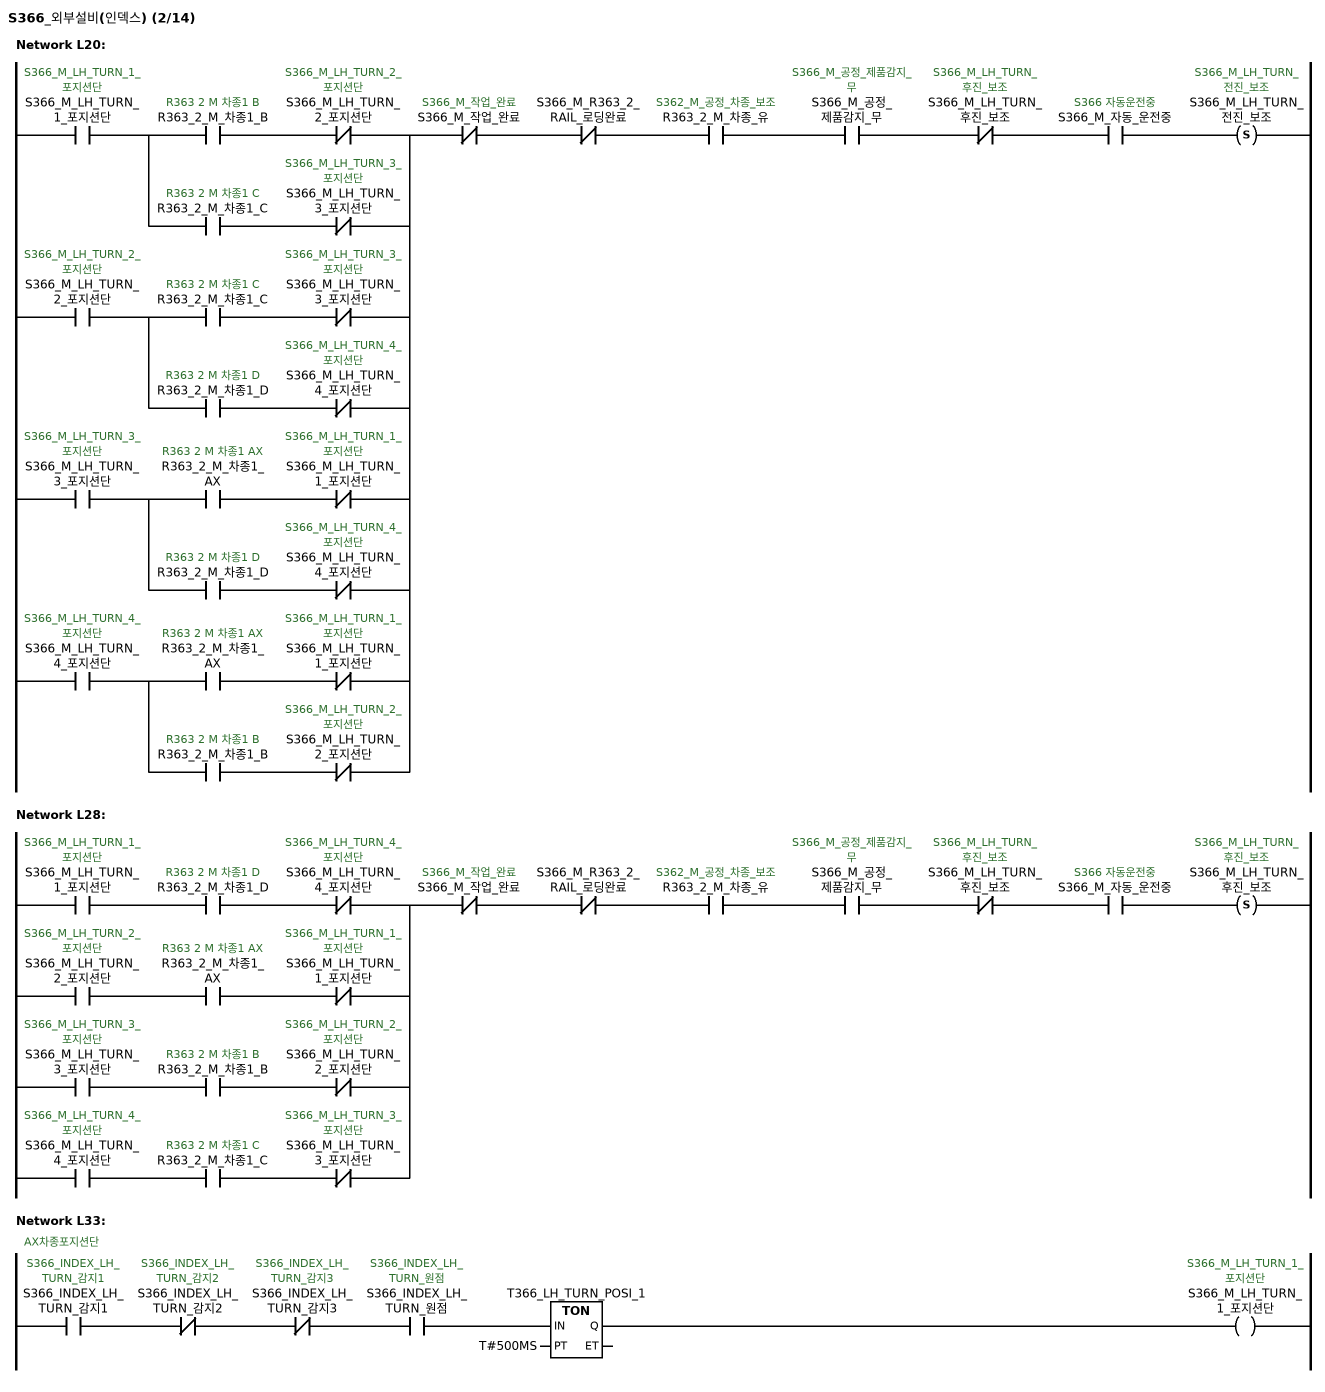
(* [picture p192: S366_외부설비(인덱스) rungs L20-L33] *)
(* Rung L20 *)
IF ((S366_M_LH_TURN_1_포지션단 AND ((R363_2_M_차종1_B AND NOT S366_M_LH_TURN_2_포지션단) OR (R363_2_M_차종1_C AND NOT S366_M_LH_TURN_3_포지션단))) OR (S366_M_LH_TURN_2_포지션단 AND ((R363_2_M_차종1_C AND NOT S366_M_LH_TURN_3_포지션단) OR (R363_2_M_차종1_D AND NOT S366_M_LH_TURN_4_포지션단))) OR (S366_M_LH_TURN_3_포지션단 AND ((R363_2_M_차종1_AX AND NOT S366_M_LH_TURN_1_포지션단) OR (R363_2_M_차종1_D AND NOT S366_M_LH_TURN_4_포지션단))) OR (S366_M_LH_TURN_4_포지션단 AND ((R363_2_M_차종1_AX AND NOT S366_M_LH_TURN_1_포지션단) OR (R363_2_M_차종1_B AND NOT S366_M_LH_TURN_2_포지션단)))) AND NOT S366_M_작업_완료 AND NOT S366_M_R363_2_RAIL_로딩완료 AND R363_2_M_차종_유 AND S366_M_공정_제품감지_무 AND NOT S366_M_LH_TURN_후진_보조 AND S366_M_자동_운전중 THEN
    S366_M_LH_TURN_전진_보조 := TRUE;
END_IF;
(* Rung L28 *)
IF ((S366_M_LH_TURN_1_포지션단 AND R363_2_M_차종1_D AND NOT S366_M_LH_TURN_4_포지션단) OR (S366_M_LH_TURN_2_포지션단 AND R363_2_M_차종1_AX AND NOT S366_M_LH_TURN_1_포지션단) OR (S366_M_LH_TURN_3_포지션단 AND R363_2_M_차종1_B AND NOT S366_M_LH_TURN_2_포지션단) OR (S366_M_LH_TURN_4_포지션단 AND R363_2_M_차종1_C AND NOT S366_M_LH_TURN_3_포지션단)) AND NOT S366_M_작업_완료 AND NOT S366_M_R363_2_RAIL_로딩완료 AND R363_2_M_차종_유 AND S366_M_공정_제품감지_무 AND NOT S366_M_LH_TURN_후진_보조 AND S366_M_자동_운전중 THEN
    S366_M_LH_TURN_후진_보조 := TRUE;
END_IF;
(* AX차종포지션단 *)
(* Rung L33 *)
T366_LH_TURN_POSI_1(IN := S366_INDEX_LH_TURN_감지1 AND NOT S366_INDEX_LH_TURN_감지2 AND NOT S366_INDEX_LH_TURN_감지3 AND S366_INDEX_LH_TURN_원점, PT := T#500MS);
S366_M_LH_TURN_1_포지션단 := T366_LH_TURN_POSI_1.Q;

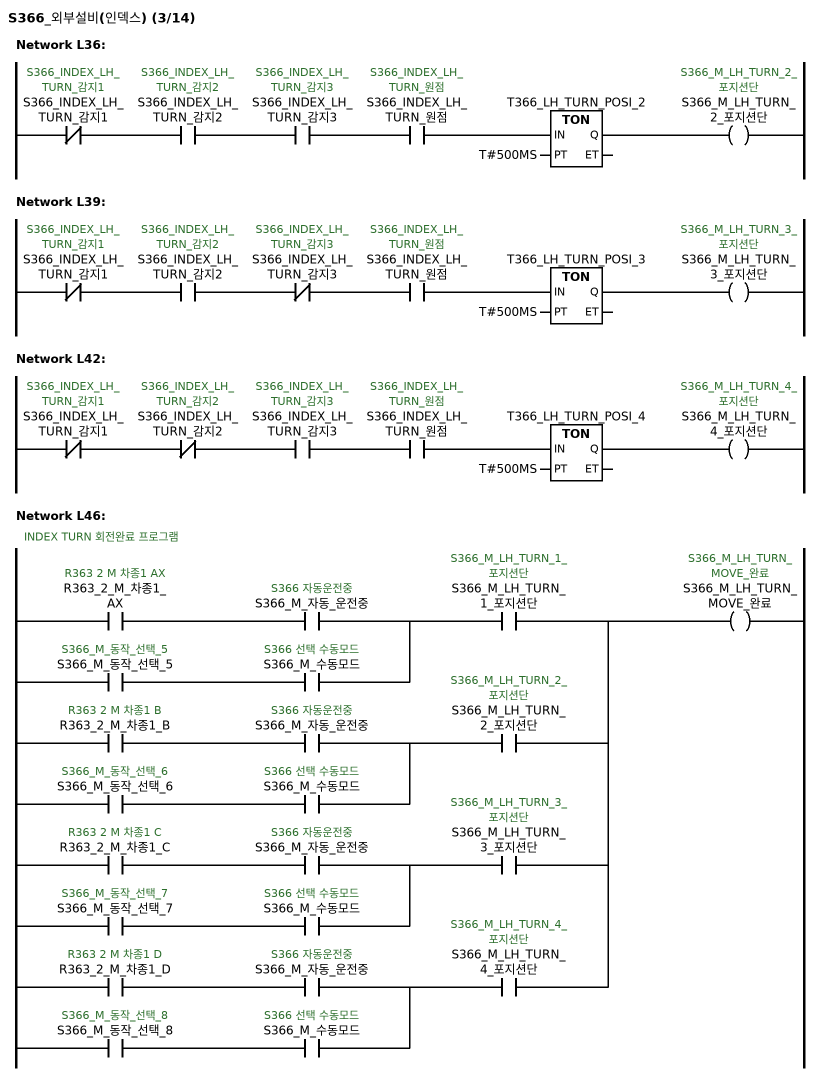
(* Rung L36 *)
T366_LH_TURN_POSI_2(IN := NOT S366_INDEX_LH_TURN_감지1 AND S366_INDEX_LH_TURN_감지2 AND S366_INDEX_LH_TURN_감지3 AND S366_INDEX_LH_TURN_원점, PT := T#500MS);
S366_M_LH_TURN_2_포지션단 := T366_LH_TURN_POSI_2.Q;
(* Rung L39 *)
T366_LH_TURN_POSI_3(IN := NOT S366_INDEX_LH_TURN_감지1 AND S366_INDEX_LH_TURN_감지2 AND NOT S366_INDEX_LH_TURN_감지3 AND S366_INDEX_LH_TURN_원점, PT := T#500MS);
S366_M_LH_TURN_3_포지션단 := T366_LH_TURN_POSI_3.Q;
(* Rung L42 *)
T366_LH_TURN_POSI_4(IN := NOT S366_INDEX_LH_TURN_감지1 AND NOT S366_INDEX_LH_TURN_감지2 AND S366_INDEX_LH_TURN_감지3 AND S366_INDEX_LH_TURN_원점, PT := T#500MS);
S366_M_LH_TURN_4_포지션단 := T366_LH_TURN_POSI_4.Q;
(* INDEX TURN 회전완료 프로그램 *)
(* Rung L46 *)
S366_M_LH_TURN_MOVE_완료 := (((R363_2_M_차종1_AX AND S366_M_자동_운전중) OR (S366_M_동작_선택_5 AND S366_M_수동모드)) AND S366_M_LH_TURN_1_포지션단) OR (((R363_2_M_차종1_B AND S366_M_자동_운전중) OR (S366_M_동작_선택_6 AND S366_M_수동모드)) AND S366_M_LH_TURN_2_포지션단) OR (((R363_2_M_차종1_C AND S366_M_자동_운전중) OR (S366_M_동작_선택_7 AND S366_M_수동모드)) AND S366_M_LH_TURN_3_포지션단) OR (((R363_2_M_차종1_D AND S366_M_자동_운전중) OR (S366_M_동작_선택_8 AND S366_M_수동모드)) AND S366_M_LH_TURN_4_포지션단);

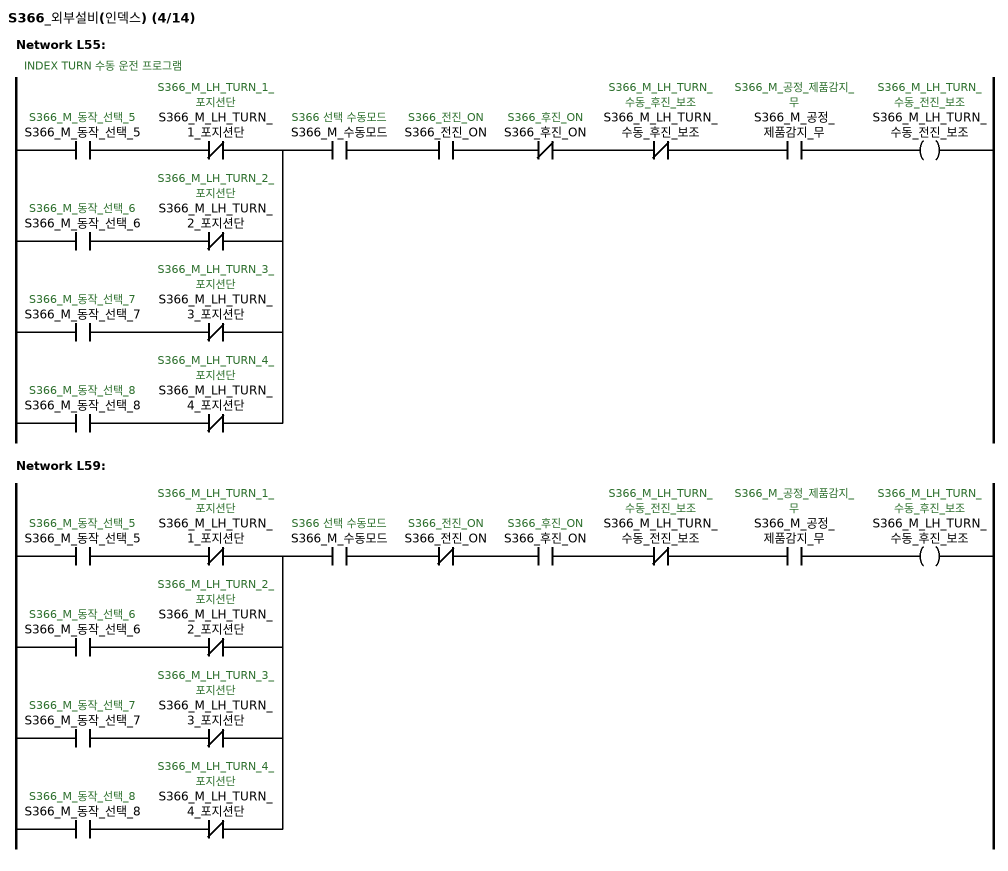
(* INDEX TURN 수동 운전 프로그램 *)
(* Rung L55 *)
S366_M_LH_TURN_수동_전진_보조 := ((S366_M_동작_선택_5 AND NOT S366_M_LH_TURN_1_포지션단) OR (S366_M_동작_선택_6 AND NOT S366_M_LH_TURN_2_포지션단) OR (S366_M_동작_선택_7 AND NOT S366_M_LH_TURN_3_포지션단) OR (S366_M_동작_선택_8 AND NOT S366_M_LH_TURN_4_포지션단)) AND S366_M_수동모드 AND S366_전진_ON AND NOT S366_후진_ON AND NOT S366_M_LH_TURN_수동_후진_보조 AND S366_M_공정_제품감지_무;
(* Rung L59 *)
S366_M_LH_TURN_수동_후진_보조 := ((S366_M_동작_선택_5 AND NOT S366_M_LH_TURN_1_포지션단) OR (S366_M_동작_선택_6 AND NOT S366_M_LH_TURN_2_포지션단) OR (S366_M_동작_선택_7 AND NOT S366_M_LH_TURN_3_포지션단) OR (S366_M_동작_선택_8 AND NOT S366_M_LH_TURN_4_포지션단)) AND S366_M_수동모드 AND NOT S366_전진_ON AND S366_후진_ON AND NOT S366_M_LH_TURN_수동_전진_보조 AND S366_M_공정_제품감지_무;

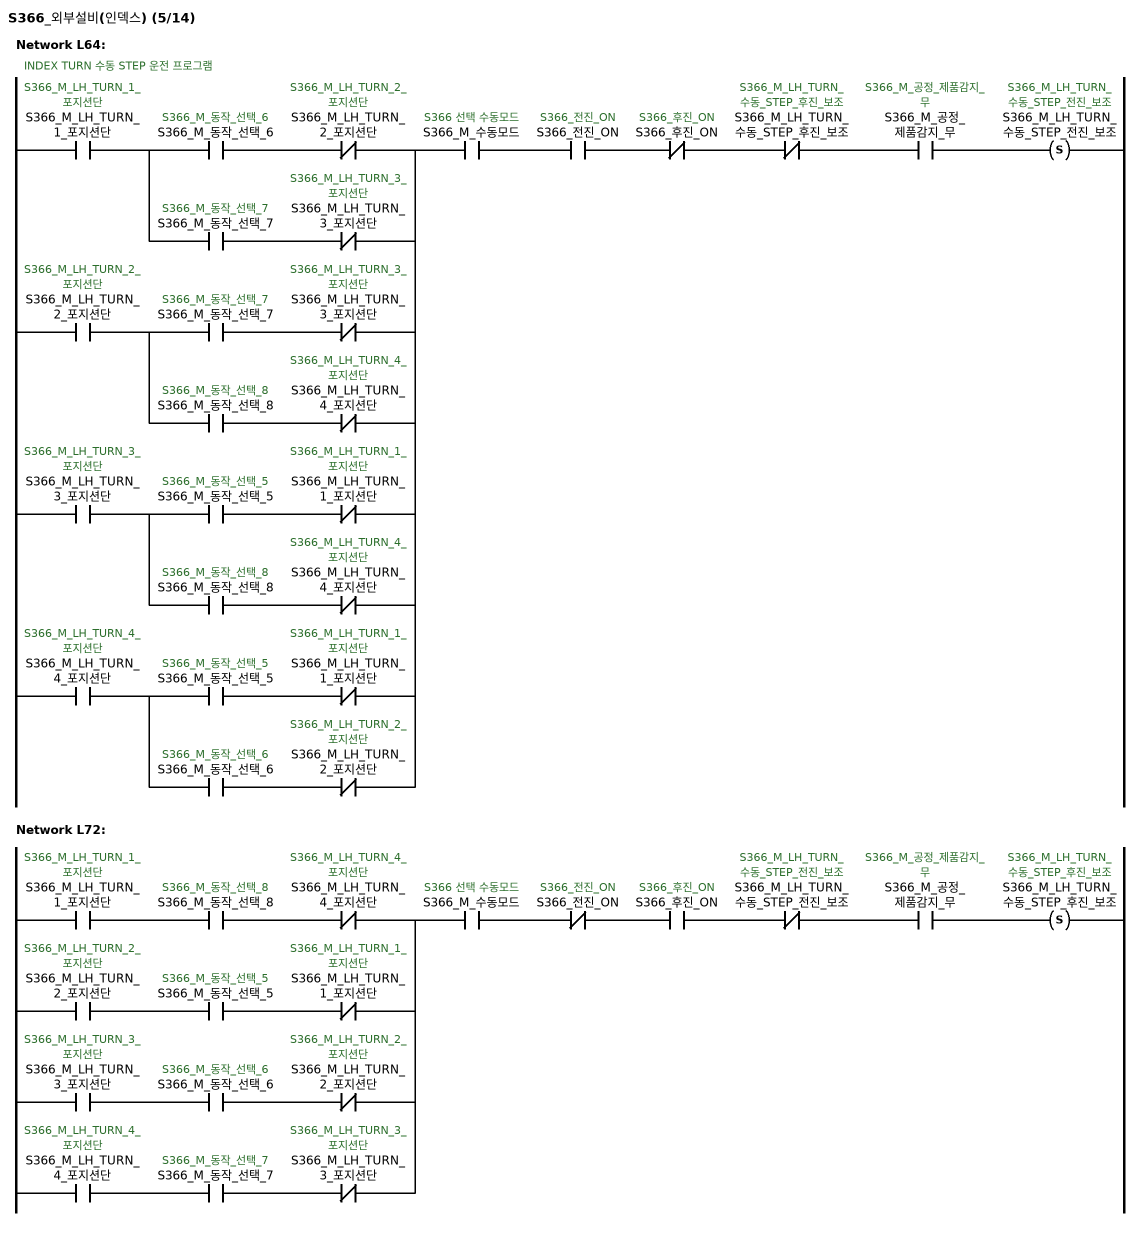
(* INDEX TURN 수동 STEP 운전 프로그램 *)
(* Rung L64 *)
IF ((S366_M_LH_TURN_1_포지션단 AND ((S366_M_동작_선택_6 AND NOT S366_M_LH_TURN_2_포지션단) OR (S366_M_동작_선택_7 AND NOT S366_M_LH_TURN_3_포지션단))) OR (S366_M_LH_TURN_2_포지션단 AND ((S366_M_동작_선택_7 AND NOT S366_M_LH_TURN_3_포지션단) OR (S366_M_동작_선택_8 AND NOT S366_M_LH_TURN_4_포지션단))) OR (S366_M_LH_TURN_3_포지션단 AND ((S366_M_동작_선택_5 AND NOT S366_M_LH_TURN_1_포지션단) OR (S366_M_동작_선택_8 AND NOT S366_M_LH_TURN_4_포지션단))) OR (S366_M_LH_TURN_4_포지션단 AND ((S366_M_동작_선택_5 AND NOT S366_M_LH_TURN_1_포지션단) OR (S366_M_동작_선택_6 AND NOT S366_M_LH_TURN_2_포지션단)))) AND S366_M_수동모드 AND S366_전진_ON AND NOT S366_후진_ON AND NOT S366_M_LH_TURN_수동_STEP_후진_보조 AND S366_M_공정_제품감지_무 THEN
    S366_M_LH_TURN_수동_STEP_전진_보조 := TRUE;
END_IF;
(* Rung L72 *)
IF ((S366_M_LH_TURN_1_포지션단 AND S366_M_동작_선택_8 AND NOT S366_M_LH_TURN_4_포지션단) OR (S366_M_LH_TURN_2_포지션단 AND S366_M_동작_선택_5 AND NOT S366_M_LH_TURN_1_포지션단) OR (S366_M_LH_TURN_3_포지션단 AND S366_M_동작_선택_6 AND NOT S366_M_LH_TURN_2_포지션단) OR (S366_M_LH_TURN_4_포지션단 AND S366_M_동작_선택_7 AND NOT S366_M_LH_TURN_3_포지션단)) AND S366_M_수동모드 AND NOT S366_전진_ON AND S366_후진_ON AND NOT S366_M_LH_TURN_수동_STEP_전진_보조 AND S366_M_공정_제품감지_무 THEN
    S366_M_LH_TURN_수동_STEP_후진_보조 := TRUE;
END_IF;

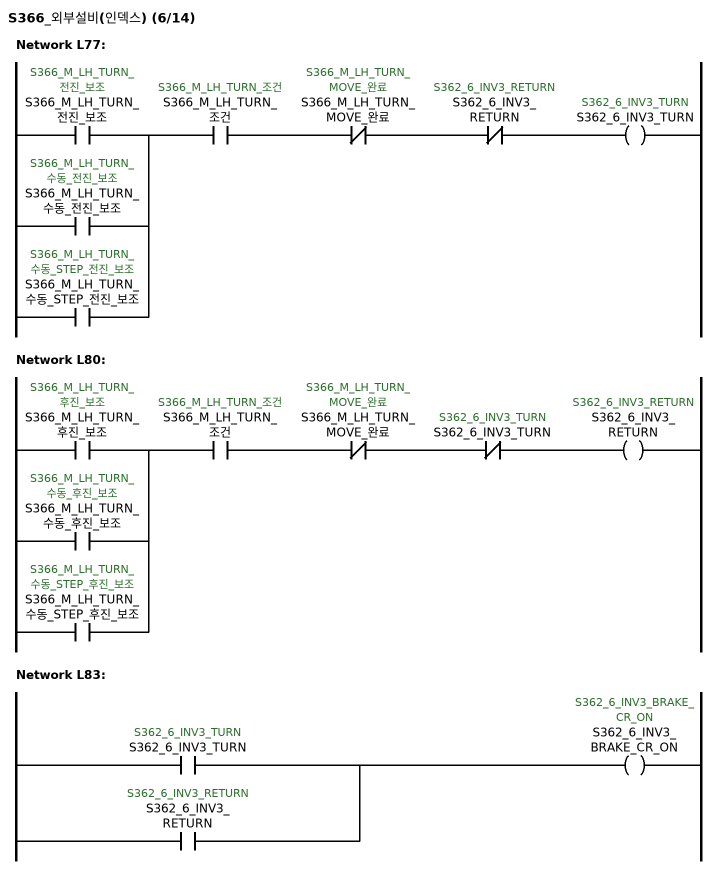
(* Rung L77 *)
S362_6_INV3_TURN := (S366_M_LH_TURN_전진_보조 OR S366_M_LH_TURN_수동_전진_보조 OR S366_M_LH_TURN_수동_STEP_전진_보조) AND S366_M_LH_TURN_조건 AND NOT S366_M_LH_TURN_MOVE_완료 AND NOT S362_6_INV3_RETURN;
(* Rung L80 *)
S362_6_INV3_RETURN := (S366_M_LH_TURN_후진_보조 OR S366_M_LH_TURN_수동_후진_보조 OR S366_M_LH_TURN_수동_STEP_후진_보조) AND S366_M_LH_TURN_조건 AND NOT S366_M_LH_TURN_MOVE_완료 AND NOT S362_6_INV3_TURN;
(* Rung L83 *)
S362_6_INV3_BRAKE_CR_ON := S362_6_INV3_TURN OR S362_6_INV3_RETURN;

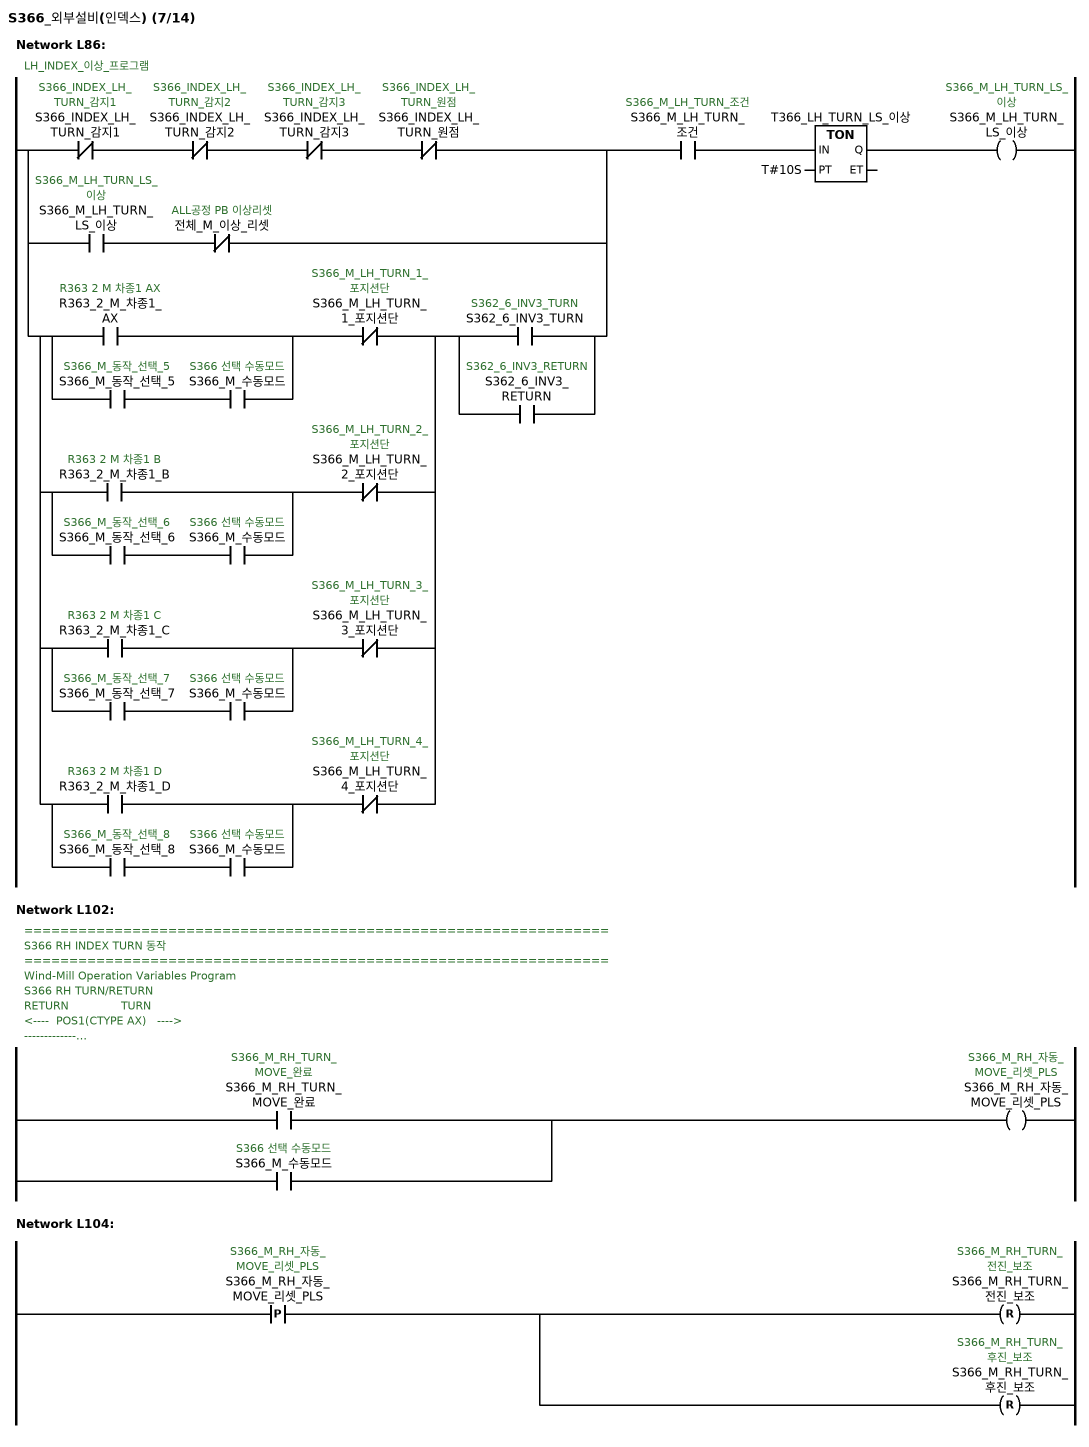
(* LH_INDEX_이상_프로그램 *)
(* Rung L86 *)
T366_LH_TURN_LS_이상(IN := ((NOT S366_INDEX_LH_TURN_감지1 AND NOT S366_INDEX_LH_TURN_감지2 AND NOT S366_INDEX_LH_TURN_감지3 AND NOT S366_INDEX_LH_TURN_원점) OR (S366_M_LH_TURN_LS_이상 AND NOT 전체_M_이상_리셋) OR ((((R363_2_M_차종1_AX OR (S366_M_동작_선택_5 AND S366_M_수동모드)) AND NOT S366_M_LH_TURN_1_포지션단) OR ((R363_2_M_차종1_B OR (S366_M_동작_선택_6 AND S366_M_수동모드)) AND NOT S366_M_LH_TURN_2_포지션단) OR ((R363_2_M_차종1_C OR (S366_M_동작_선택_7 AND S366_M_수동모드)) AND NOT S366_M_LH_TURN_3_포지션단) OR ((R363_2_M_차종1_D OR (S366_M_동작_선택_8 AND S366_M_수동모드)) AND NOT S366_M_LH_TURN_4_포지션단)) AND (S362_6_INV3_TURN OR S362_6_INV3_RETURN))) AND S366_M_LH_TURN_조건, PT := T#10S);
S366_M_LH_TURN_LS_이상 := T366_LH_TURN_LS_이상.Q;
(* ================================================================= *)
(* S366 RH INDEX TURN 동작 *)
(* ================================================================= *)
(* Wind-Mill Operation Variables Program / S366 RH TURN/RETURN *)
(* RETURN               TURN / <----  POS1(CTYPE AX)   ----> / -------------- / l              l / l              l / l              l / POS2 (CTYPE B) l              l  POS4 (CTYPE D) / l              l / l              l / l              l / -------------- / POS3 (CTYPE C) *)
(* 자동 MOVE 리셋 프로그램 *)
(* Rung L102 *)
S366_M_RH_자동_MOVE_리셋_PLS := S366_M_RH_TURN_MOVE_완료 OR S366_M_수동모드;
(* Rung L104 *)
_e3(CLK := S366_M_RH_자동_MOVE_리셋_PLS);
IF _e3.Q THEN
    S366_M_RH_TURN_전진_보조 := FALSE;
    S366_M_RH_TURN_후진_보조 := FALSE;
END_IF;

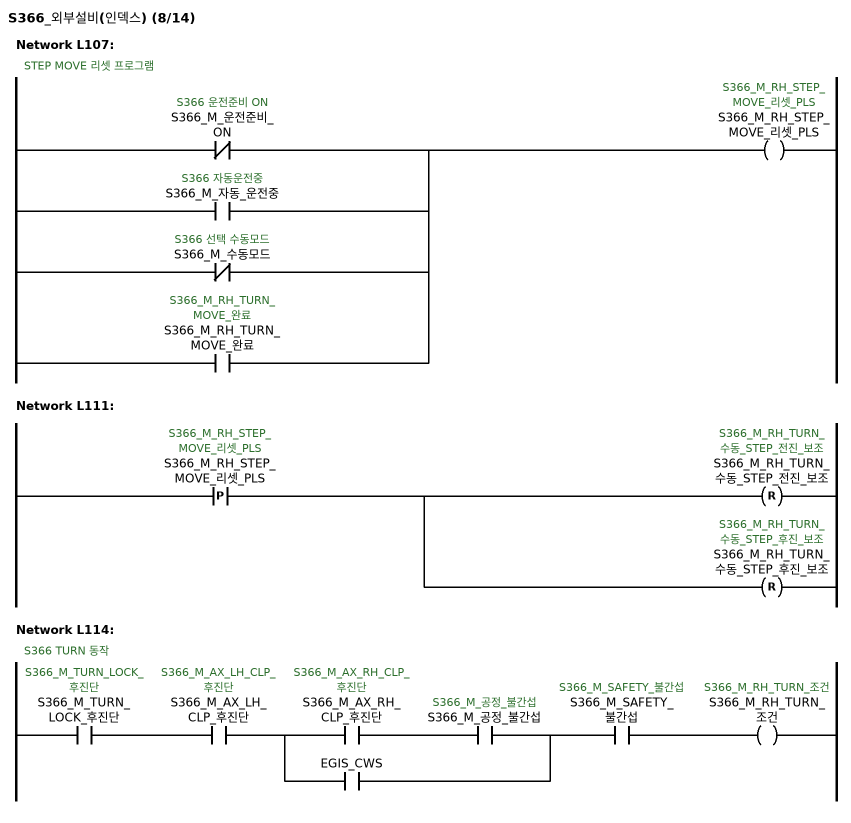
(* STEP MOVE 리셋 프로그램 *)
(* Rung L107 *)
S366_M_RH_STEP_MOVE_리셋_PLS := NOT S366_M_운전준비_ON OR S366_M_자동_운전중 OR NOT S366_M_수동모드 OR S366_M_RH_TURN_MOVE_완료;
(* Rung L111 *)
_e4(CLK := S366_M_RH_STEP_MOVE_리셋_PLS);
IF _e4.Q THEN
    S366_M_RH_TURN_수동_STEP_전진_보조 := FALSE;
    S366_M_RH_TURN_수동_STEP_후진_보조 := FALSE;
END_IF;
(* S366 TURN 동작 *)
(* Rung L114 *)
S366_M_RH_TURN_조건 := S366_M_TURN_LOCK_후진단 AND S366_M_AX_LH_CLP_후진단 AND ((S366_M_AX_RH_CLP_후진단 AND S366_M_공정_불간섭) OR EGIS_CWS) AND S366_M_SAFETY_불간섭;

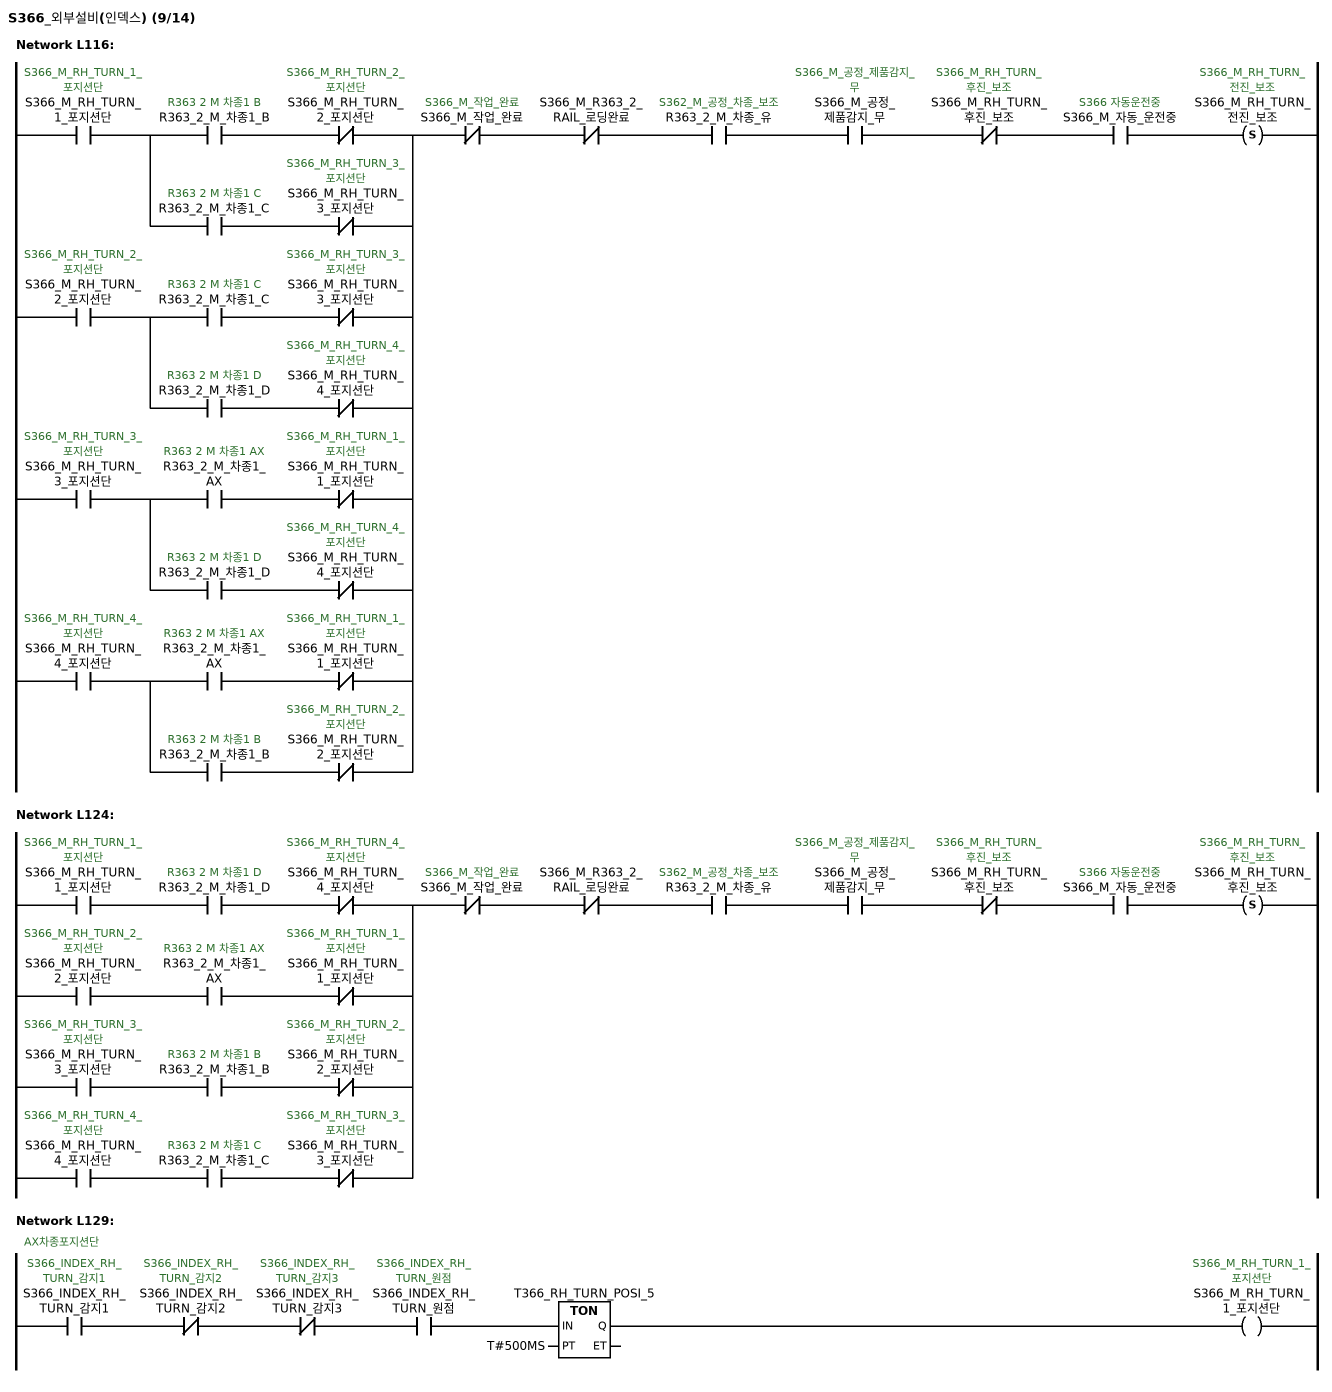
(* Rung L116 *)
IF ((S366_M_RH_TURN_1_포지션단 AND ((R363_2_M_차종1_B AND NOT S366_M_RH_TURN_2_포지션단) OR (R363_2_M_차종1_C AND NOT S366_M_RH_TURN_3_포지션단))) OR (S366_M_RH_TURN_2_포지션단 AND ((R363_2_M_차종1_C AND NOT S366_M_RH_TURN_3_포지션단) OR (R363_2_M_차종1_D AND NOT S366_M_RH_TURN_4_포지션단))) OR (S366_M_RH_TURN_3_포지션단 AND ((R363_2_M_차종1_AX AND NOT S366_M_RH_TURN_1_포지션단) OR (R363_2_M_차종1_D AND NOT S366_M_RH_TURN_4_포지션단))) OR (S366_M_RH_TURN_4_포지션단 AND ((R363_2_M_차종1_AX AND NOT S366_M_RH_TURN_1_포지션단) OR (R363_2_M_차종1_B AND NOT S366_M_RH_TURN_2_포지션단)))) AND NOT S366_M_작업_완료 AND NOT S366_M_R363_2_RAIL_로딩완료 AND R363_2_M_차종_유 AND S366_M_공정_제품감지_무 AND NOT S366_M_RH_TURN_후진_보조 AND S366_M_자동_운전중 THEN
    S366_M_RH_TURN_전진_보조 := TRUE;
END_IF;
(* Rung L124 *)
IF ((S366_M_RH_TURN_1_포지션단 AND R363_2_M_차종1_D AND NOT S366_M_RH_TURN_4_포지션단) OR (S366_M_RH_TURN_2_포지션단 AND R363_2_M_차종1_AX AND NOT S366_M_RH_TURN_1_포지션단) OR (S366_M_RH_TURN_3_포지션단 AND R363_2_M_차종1_B AND NOT S366_M_RH_TURN_2_포지션단) OR (S366_M_RH_TURN_4_포지션단 AND R363_2_M_차종1_C AND NOT S366_M_RH_TURN_3_포지션단)) AND NOT S366_M_작업_완료 AND NOT S366_M_R363_2_RAIL_로딩완료 AND R363_2_M_차종_유 AND S366_M_공정_제품감지_무 AND NOT S366_M_RH_TURN_후진_보조 AND S366_M_자동_운전중 THEN
    S366_M_RH_TURN_후진_보조 := TRUE;
END_IF;
(* AX차종포지션단 *)
(* Rung L129 *)
T366_RH_TURN_POSI_5(IN := S366_INDEX_RH_TURN_감지1 AND NOT S366_INDEX_RH_TURN_감지2 AND NOT S366_INDEX_RH_TURN_감지3 AND S366_INDEX_RH_TURN_원점, PT := T#500MS);
S366_M_RH_TURN_1_포지션단 := T366_RH_TURN_POSI_5.Q;

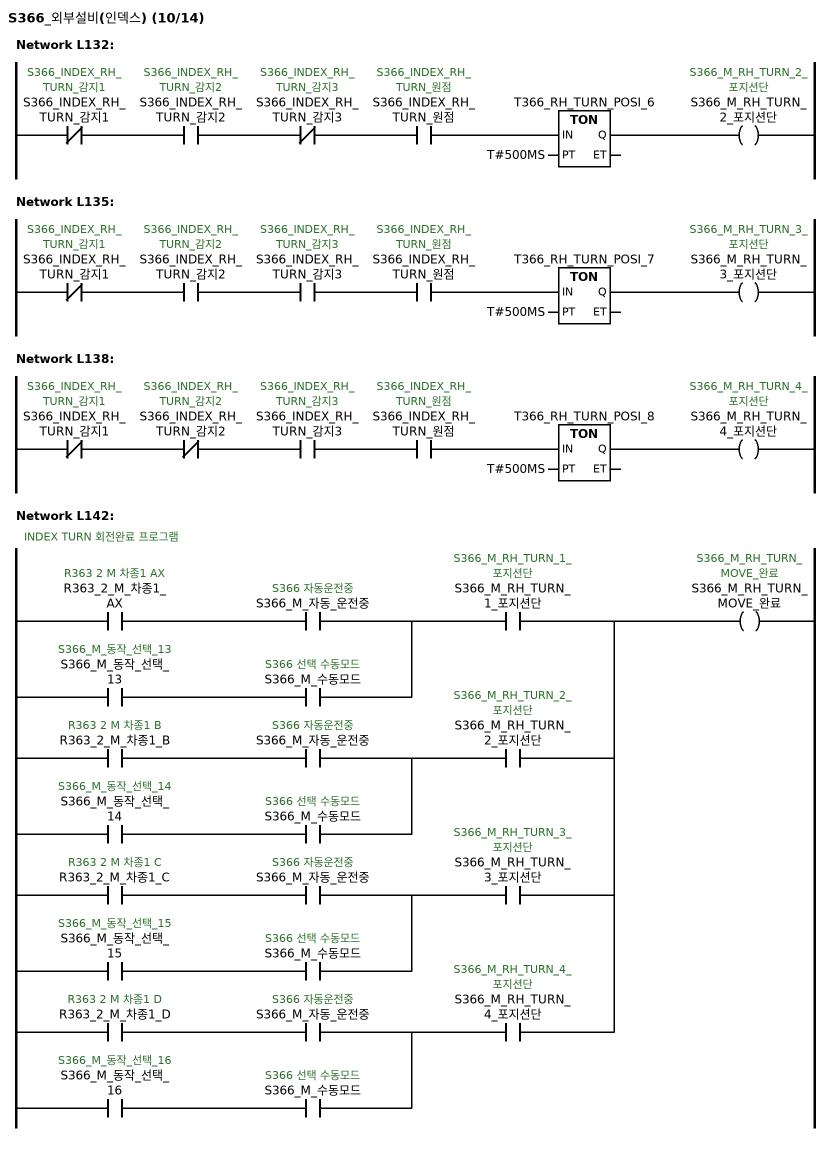
(* Rung L132 *)
T366_RH_TURN_POSI_6(IN := NOT S366_INDEX_RH_TURN_감지1 AND S366_INDEX_RH_TURN_감지2 AND NOT S366_INDEX_RH_TURN_감지3 AND S366_INDEX_RH_TURN_원점, PT := T#500MS);
S366_M_RH_TURN_2_포지션단 := T366_RH_TURN_POSI_6.Q;
(* Rung L135 *)
T366_RH_TURN_POSI_7(IN := NOT S366_INDEX_RH_TURN_감지1 AND S366_INDEX_RH_TURN_감지2 AND S366_INDEX_RH_TURN_감지3 AND S366_INDEX_RH_TURN_원점, PT := T#500MS);
S366_M_RH_TURN_3_포지션단 := T366_RH_TURN_POSI_7.Q;
(* Rung L138 *)
T366_RH_TURN_POSI_8(IN := NOT S366_INDEX_RH_TURN_감지1 AND NOT S366_INDEX_RH_TURN_감지2 AND S366_INDEX_RH_TURN_감지3 AND S366_INDEX_RH_TURN_원점, PT := T#500MS);
S366_M_RH_TURN_4_포지션단 := T366_RH_TURN_POSI_8.Q;
(* INDEX TURN 회전완료 프로그램 *)
(* Rung L142 *)
S366_M_RH_TURN_MOVE_완료 := (((R363_2_M_차종1_AX AND S366_M_자동_운전중) OR (S366_M_동작_선택_13 AND S366_M_수동모드)) AND S366_M_RH_TURN_1_포지션단) OR (((R363_2_M_차종1_B AND S366_M_자동_운전중) OR (S366_M_동작_선택_14 AND S366_M_수동모드)) AND S366_M_RH_TURN_2_포지션단) OR (((R363_2_M_차종1_C AND S366_M_자동_운전중) OR (S366_M_동작_선택_15 AND S366_M_수동모드)) AND S366_M_RH_TURN_3_포지션단) OR (((R363_2_M_차종1_D AND S366_M_자동_운전중) OR (S366_M_동작_선택_16 AND S366_M_수동모드)) AND S366_M_RH_TURN_4_포지션단);

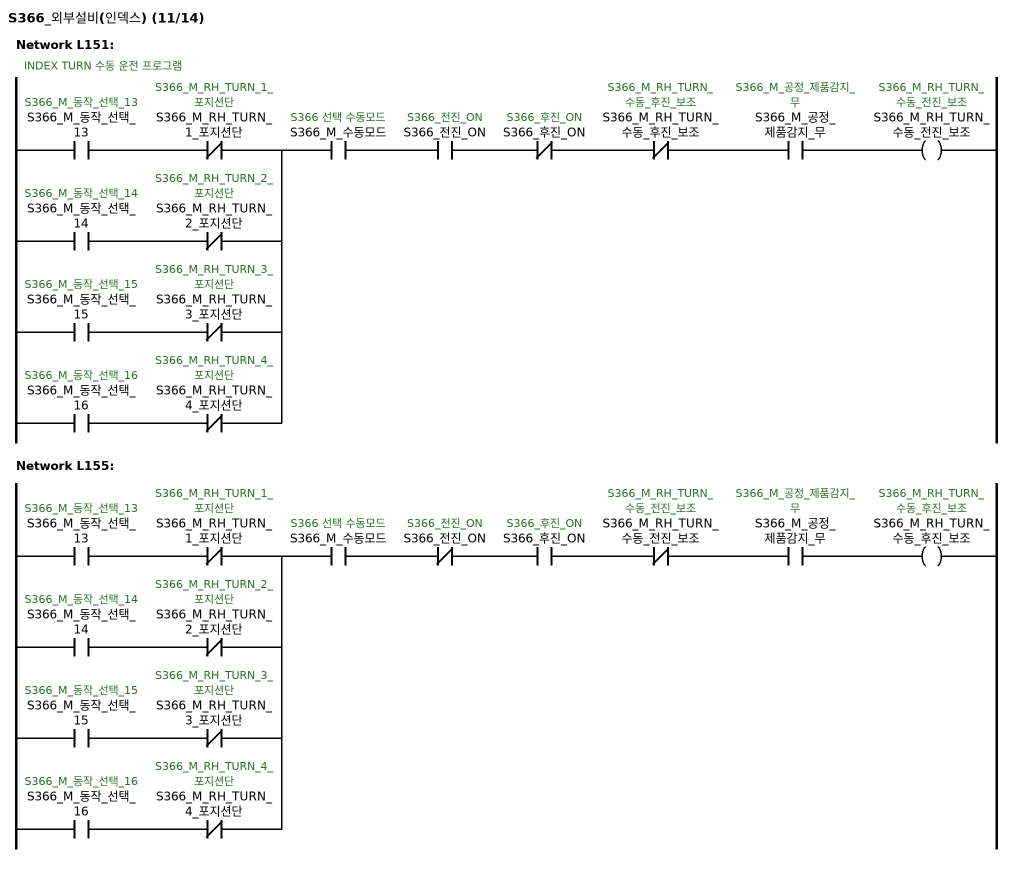
(* INDEX TURN 수동 운전 프로그램 *)
(* Rung L151 *)
S366_M_RH_TURN_수동_전진_보조 := ((S366_M_동작_선택_13 AND NOT S366_M_RH_TURN_1_포지션단) OR (S366_M_동작_선택_14 AND NOT S366_M_RH_TURN_2_포지션단) OR (S366_M_동작_선택_15 AND NOT S366_M_RH_TURN_3_포지션단) OR (S366_M_동작_선택_16 AND NOT S366_M_RH_TURN_4_포지션단)) AND S366_M_수동모드 AND S366_전진_ON AND NOT S366_후진_ON AND NOT S366_M_RH_TURN_수동_후진_보조 AND S366_M_공정_제품감지_무;
(* Rung L155 *)
S366_M_RH_TURN_수동_후진_보조 := ((S366_M_동작_선택_13 AND NOT S366_M_RH_TURN_1_포지션단) OR (S366_M_동작_선택_14 AND NOT S366_M_RH_TURN_2_포지션단) OR (S366_M_동작_선택_15 AND NOT S366_M_RH_TURN_3_포지션단) OR (S366_M_동작_선택_16 AND NOT S366_M_RH_TURN_4_포지션단)) AND S366_M_수동모드 AND NOT S366_전진_ON AND S366_후진_ON AND NOT S366_M_RH_TURN_수동_전진_보조 AND S366_M_공정_제품감지_무;

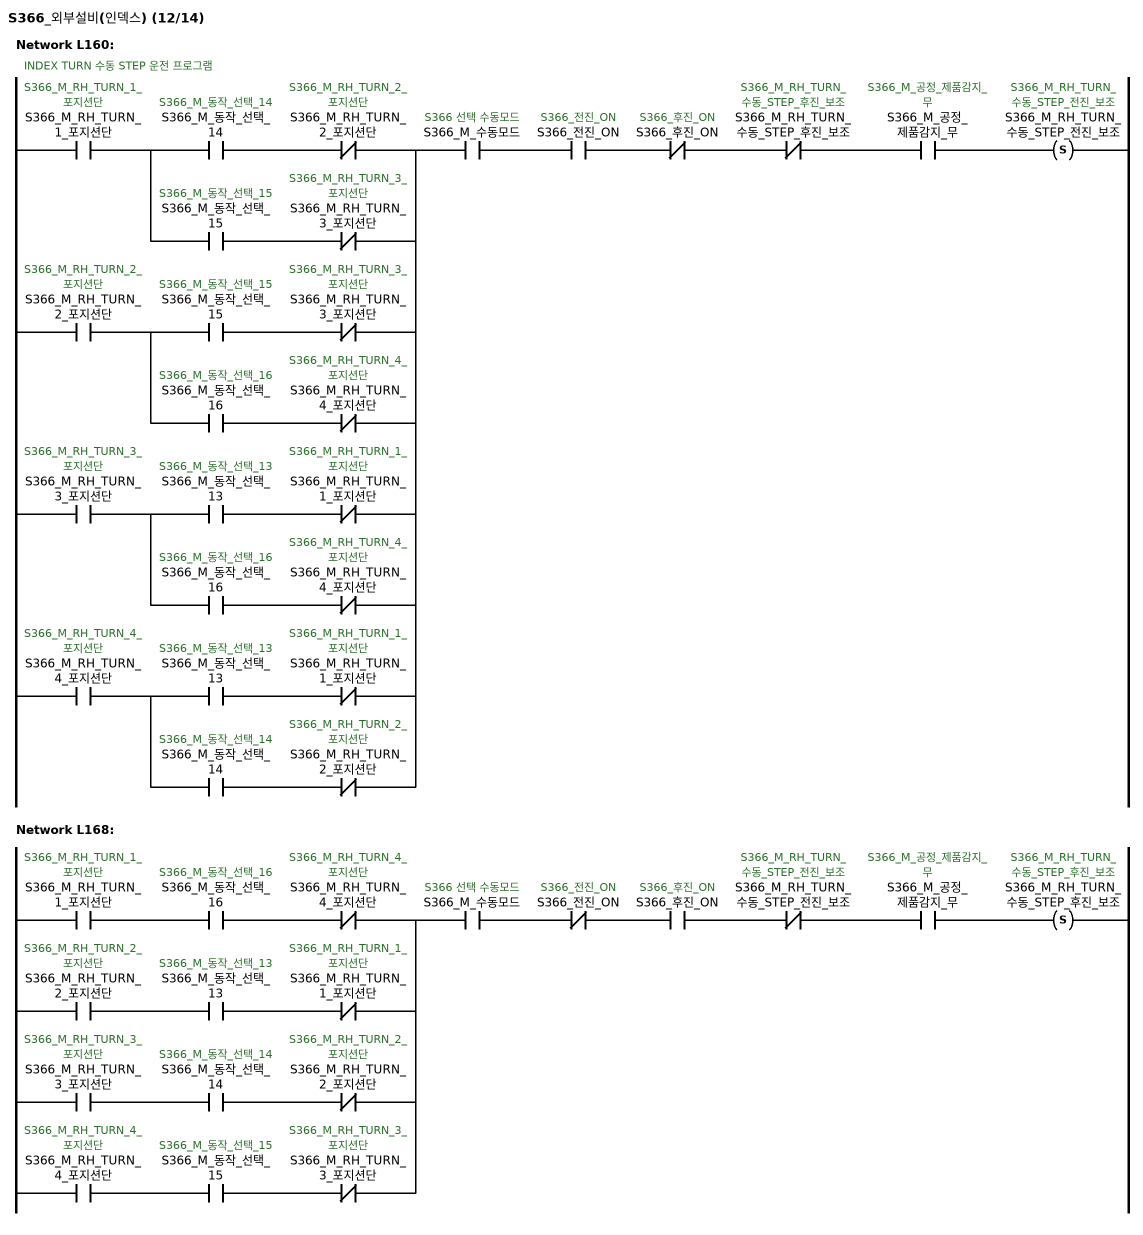
(* INDEX TURN 수동 STEP 운전 프로그램 *)
(* Rung L160 *)
IF ((S366_M_RH_TURN_1_포지션단 AND ((S366_M_동작_선택_14 AND NOT S366_M_RH_TURN_2_포지션단) OR (S366_M_동작_선택_15 AND NOT S366_M_RH_TURN_3_포지션단))) OR (S366_M_RH_TURN_2_포지션단 AND ((S366_M_동작_선택_15 AND NOT S366_M_RH_TURN_3_포지션단) OR (S366_M_동작_선택_16 AND NOT S366_M_RH_TURN_4_포지션단))) OR (S366_M_RH_TURN_3_포지션단 AND ((S366_M_동작_선택_13 AND NOT S366_M_RH_TURN_1_포지션단) OR (S366_M_동작_선택_16 AND NOT S366_M_RH_TURN_4_포지션단))) OR (S366_M_RH_TURN_4_포지션단 AND ((S366_M_동작_선택_13 AND NOT S366_M_RH_TURN_1_포지션단) OR (S366_M_동작_선택_14 AND NOT S366_M_RH_TURN_2_포지션단)))) AND S366_M_수동모드 AND S366_전진_ON AND NOT S366_후진_ON AND NOT S366_M_RH_TURN_수동_STEP_후진_보조 AND S366_M_공정_제품감지_무 THEN
    S366_M_RH_TURN_수동_STEP_전진_보조 := TRUE;
END_IF;
(* Rung L168 *)
IF ((S366_M_RH_TURN_1_포지션단 AND S366_M_동작_선택_16 AND NOT S366_M_RH_TURN_4_포지션단) OR (S366_M_RH_TURN_2_포지션단 AND S366_M_동작_선택_13 AND NOT S366_M_RH_TURN_1_포지션단) OR (S366_M_RH_TURN_3_포지션단 AND S366_M_동작_선택_14 AND NOT S366_M_RH_TURN_2_포지션단) OR (S366_M_RH_TURN_4_포지션단 AND S366_M_동작_선택_15 AND NOT S366_M_RH_TURN_3_포지션단)) AND S366_M_수동모드 AND NOT S366_전진_ON AND S366_후진_ON AND NOT S366_M_RH_TURN_수동_STEP_전진_보조 AND S366_M_공정_제품감지_무 THEN
    S366_M_RH_TURN_수동_STEP_후진_보조 := TRUE;
END_IF;

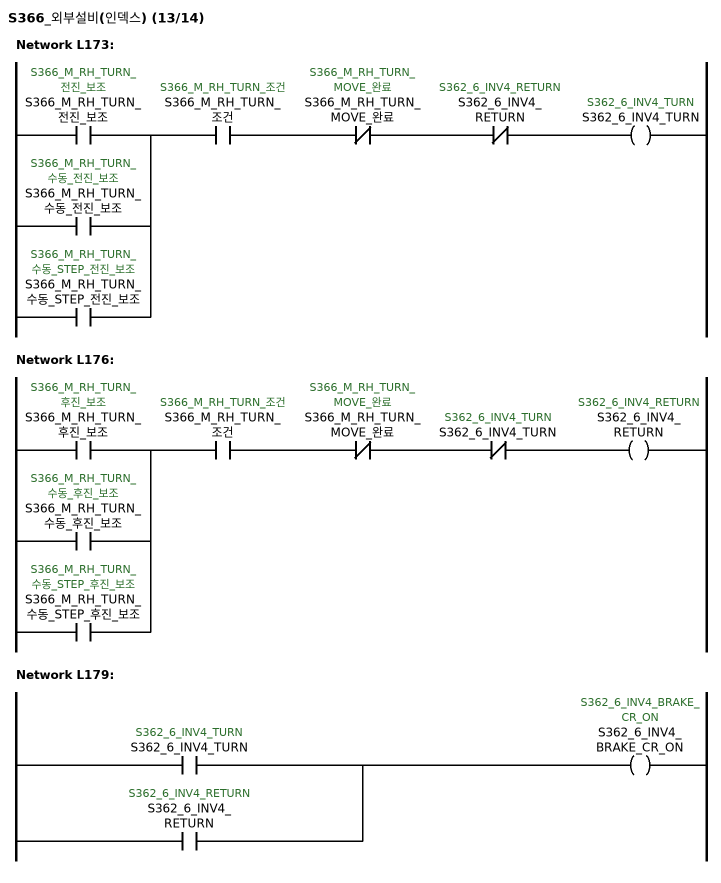
(* Rung L173 *)
S362_6_INV4_TURN := (S366_M_RH_TURN_전진_보조 OR S366_M_RH_TURN_수동_전진_보조 OR S366_M_RH_TURN_수동_STEP_전진_보조) AND S366_M_RH_TURN_조건 AND NOT S366_M_RH_TURN_MOVE_완료 AND NOT S362_6_INV4_RETURN;
(* Rung L176 *)
S362_6_INV4_RETURN := (S366_M_RH_TURN_후진_보조 OR S366_M_RH_TURN_수동_후진_보조 OR S366_M_RH_TURN_수동_STEP_후진_보조) AND S366_M_RH_TURN_조건 AND NOT S366_M_RH_TURN_MOVE_완료 AND NOT S362_6_INV4_TURN;
(* Rung L179 *)
S362_6_INV4_BRAKE_CR_ON := S362_6_INV4_TURN OR S362_6_INV4_RETURN;

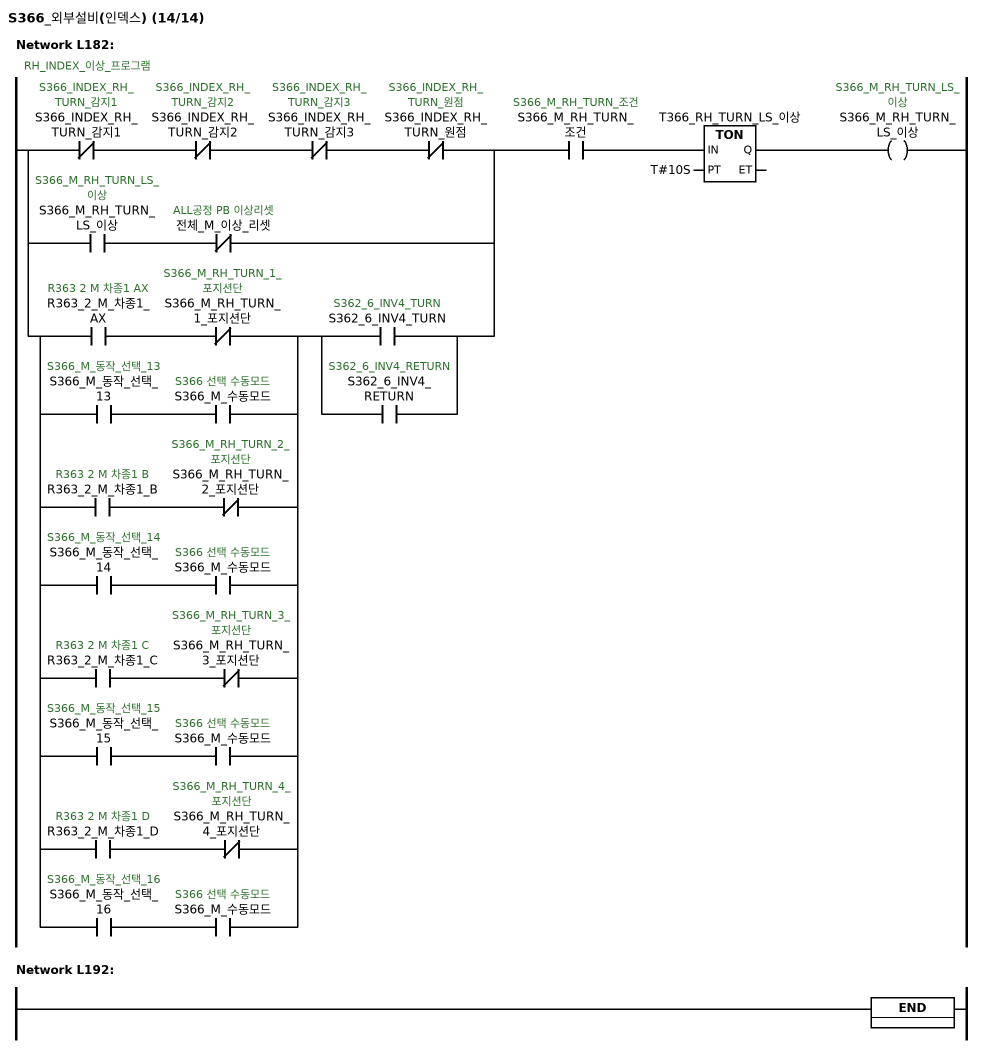
(* RH_INDEX_이상_프로그램 *)
(* Rung L182 *)
T366_RH_TURN_LS_이상(IN := ((NOT S366_INDEX_RH_TURN_감지1 AND NOT S366_INDEX_RH_TURN_감지2 AND NOT S366_INDEX_RH_TURN_감지3 AND NOT S366_INDEX_RH_TURN_원점) OR (S366_M_RH_TURN_LS_이상 AND NOT 전체_M_이상_리셋) OR (((R363_2_M_차종1_AX AND NOT S366_M_RH_TURN_1_포지션단) OR (S366_M_동작_선택_13 AND S366_M_수동모드) OR (R363_2_M_차종1_B AND NOT S366_M_RH_TURN_2_포지션단) OR (S366_M_동작_선택_14 AND S366_M_수동모드) OR (R363_2_M_차종1_C AND NOT S366_M_RH_TURN_3_포지션단) OR (S366_M_동작_선택_15 AND S366_M_수동모드) OR (R363_2_M_차종1_D AND NOT S366_M_RH_TURN_4_포지션단) OR (S366_M_동작_선택_16 AND S366_M_수동모드)) AND (S362_6_INV4_TURN OR S362_6_INV4_RETURN))) AND S366_M_RH_TURN_조건, PT := T#10S);
S366_M_RH_TURN_LS_이상 := T366_RH_TURN_LS_이상.Q;
(* Rung L192 *)
END();
END_PROGRAM

PROGRAM S366_로보트 (* task: 스캔 프로그램 *)
VAR_EXTERNAL RETAIN
    ALWAYS_ON : BOOL; (* AT %MW3.1 *) (* 항시 ON *)
    MCP_M_부저_정지 : BOOL; (* AT %MW350.5 *) (* MCP 부저정지 *)
    MCP_M_비상정지 : BOOL; (* AT %MW350.7 *) (* MCP 비상정지 이상 *)
    S366_M_R366_1_용접가능 : BOOL; (* AT %MW3004.10 *)
    S366_M_공정_제품감지_유 : BOOL; (* AT %MW3001.6 *) (* S366_M_공정_제품감지_유 *)
    S366_M_공정_차종_AX : BOOL; (* AT %MW3002.3 *) (* S366_M_공정_차종_AX *)
    S366_M_공정_차종_유 : BOOL; (* AT %MW3002.0 *) (* S366_M_공정_차종_유 *)
    S366_M_수동모드 : BOOL; (* AT %MW3000.3 *) (* S366 선택 수동모드 *)
    S366_M_자동_START : BOOL; (* AT %MW3000.5 *) (* S366 자동운전중 *)
    S366_M_자동_운전중 : BOOL; (* AT %MW3000.4 *) (* S366 자동운전중 *)
    S366_M_작업_완료 : BOOL; (* AT %MW3001.0 *) (* S366_M_작업_완료 *)
    S366_M_작업완료_SET_PLS : BOOL; (* AT %MW3000.8 *) (* S366 M 작업완료 SET PLS *)
    S366_M_작업완료_리셋_PLS : BOOL; (* AT %MW3000.9 *) (* S366 M 작업완료 리셋 PLS *)
    S366_M_차종1_AX : BOOL; (* AT %MW10161.0 *) (* S366 M 차종1 AX *)
    S366_M_총괄_이상 : BOOL; (* AT %MW3009.0 *) (* S366_M_총괄_이상 *)
    S367_M_R366_1_용접가능 : BOOL; (* AT %MW3504.9 *)
    S367_M_공정_제품감지_무 : BOOL; (* AT %MW3501.6 *) (* S367_M_공정_제품감지_무 *)
    S367_M_공정_제품감지_유 : BOOL; (* AT %MW3501.5 *) (* S367_M_공정_제품감지_유 *)
    S367_M_공정_차종_무 : BOOL; (* AT %MW3502.1 *) (* S367_M_공정_차종_무 *)
    S367_M_공정_차종_유 : BOOL; (* AT %MW3502.0 *) (* S367_M_공정_차종_유 *)
    S367_M_자동_운전중 : BOOL; (* AT %MW3500.4 *) (* S367 자동운전중 *)
    S367_M_작업_완료 : BOOL; (* AT %MW3501.0 *) (* S367_M_작업_완료 *)
    S367_M_차종1_AX : BOOL; (* AT %MW10181.0 *) (* S367 M 차종1 AX *)
    전체_M_GATE_비상정지_정상 : BOOL; (* AT %MW308.4 *) (* 전체 M GATE 비상정지 정상 *)
    전체_M_GATE_자동기동 : BOOL; (* AT %MW308.1 *) (* 전체_M_자동_운전 *)
    전체_M_운전준비_보조 : BOOL; (* AT %MW308.5 *)
    전체_M_이상_리셋 : BOOL; (* AT %MW308.2 *) (* ALL공정 PB 이상리셋 *)
    전체_공정_M_총괄_비상정지_정상 : BOOL; (* AT %MW304.1 *)
END_VAR
VAR
    INST1 : FB494_Robot_Hyundai_HMMI_v1;
    R366_1_M_RB_PROG_NO : INT;
    로보트제외 : BOOL;
END_VAR
VAR_EXTERNAL
    MCP_PBL_운전준비_ON : BOOL; (* AT %MW87630.0 *) (* MCP_PBL_운전준비_ON *)
    R361_1_M_I_RB_간섭무_1 : BOOL; (* AT %MW20012.0 *) (* R361_1_M_I_RB_간섭무_1 *)
    R363_2_M_I_RB_간섭무_1 : BOOL; (* AT %MW20042.0 *) (* R363_2_M_I_RB_간섭무_1 *)
    R366_1_I_RB_INPUT : ARRAY[0..3] OF WORD; (* AT %MW84060 *) (* R366_1_I_RB_INPUT *)
    R366_1_M_I_RB_1차_작업완료 : BOOL; (* AT %MW20061.2 *) (* R366_1_M_I_RB_1차_작업완료 *)
    R366_1_M_I_RB_2차_작업완료 : BOOL; (* AT %MW20061.3 *) (* R366_1_M_I_RB_2차_작업완료 *)
    R366_1_M_I_RB_3차_작업완료 : BOOL; (* AT %MW20061.4 *) (* R366_1_M_I_RB_3차_작업완료 *)
    R366_1_M_I_RB_4차_작업완료 : BOOL; (* AT %MW20061.5 *) (* R366_1_M_I_RB_4차_작업완료 *)
    R366_1_M_I_RB_5차_작업완료 : BOOL; (* AT %MW20061.6 *) (* R366_1_M_I_RB_5차_작업완료 *)
    R366_1_M_I_RB_6차_작업완료 : BOOL; (* AT %MW20061.7 *) (* R366_1_M_I_RB_6차_작업완료 *)
    R366_1_M_I_RB_7차_작업완료 : BOOL; (* AT %MW20061.8 *) (* R366_1_M_I_RB_7차_작업완료 *)
    R366_1_M_I_RB_PAUSE_보조 : BOOL; (* AT %MW20060.5 *) (* R366_1_M_I_RB_PAUSE_보조 *)
    R366_1_M_I_RB_PLC_RUN_CHK_이상 : BOOL; (* AT %MW20060.7 *) (* R366_1_M_I_RB_PLC_RUN_CHK_이상 *)
    R366_1_M_I_RB_간섭무_1 : BOOL; (* AT %MW20062.0 *) (* R366_1_M_I_RB_간섭무_1 *)
    R366_1_M_I_RB_간섭무_10 : BOOL; (* AT %MW20062.9 *) (* R366_1_M_I_RB_간섭무_10 *)
    R366_1_M_I_RB_간섭무_11 : BOOL; (* AT %MW20062.10 *) (* R366_1_M_I_RB_간섭무_11 *)
    R366_1_M_I_RB_간섭무_12 : BOOL; (* AT %MW20062.11 *) (* R366_1_M_I_RB_간섭무_12 *)
    R366_1_M_I_RB_간섭무_2 : BOOL; (* AT %MW20062.1 *) (* R366_1_M_I_RB_간섭무_2 *)
    R366_1_M_I_RB_간섭무_3 : BOOL; (* AT %MW20062.2 *) (* R366_1_M_I_RB_간섭무_3 *)
    R366_1_M_I_RB_간섭무_4 : BOOL; (* AT %MW20062.3 *) (* R366_1_M_I_RB_간섭무_4 *)
    R366_1_M_I_RB_간섭무_5 : BOOL; (* AT %MW20062.4 *) (* R366_1_M_I_RB_간섭무_5 *)
    R366_1_M_I_RB_간섭무_6 : BOOL; (* AT %MW20062.5 *) (* R366_1_M_I_RB_간섭무_6 *)
    R366_1_M_I_RB_간섭무_7 : BOOL; (* AT %MW20062.6 *) (* R366_1_M_I_RB_간섭무_7 *)
    R366_1_M_I_RB_간섭무_8 : BOOL; (* AT %MW20062.7 *) (* R366_1_M_I_RB_간섭무_8 *)
    R366_1_M_I_RB_간섭무_9 : BOOL; (* AT %MW20062.8 *) (* R366_1_M_I_RB_간섭무_9 *)
    R366_1_M_I_RB_비상정지 : BOOL; (* AT %MW20060.4 *) (* R366_1_M_I_RB_비상정지 *)
    R366_1_M_I_RB_운전준비 : BOOL; (* AT %MW20060.0 *) (* R366_1_M_I_RB_운전준비 *)
    R366_1_M_I_RB_원위치 : BOOL; (* AT %MW20060.3 *) (* R366_1_M_I_RB_원위치 *)
    R366_1_M_I_RB_이상 : BOOL; (* AT %MW20060.2 *) (* R366_1_M_I_RB_이상 *)
    R366_1_M_I_RB_자동 : BOOL; (* AT %MW20060.1 *) (* R366_1_M_I_RB_자동 *)
    R366_1_M_I_RB_최종작업완료 : BOOL; (* AT %MW20061.0 *) (* R366_1_M_I_RB_최종작업완료 *)
    R366_1_M_I_RB_프로그램_이상 : BOOL; (* AT %MW20060.6 *) (* R366_1_M_I_RB_프로그램_이상 *)
    R366_1_M_O_RB_1_CYCLE_SET : BOOL; (* AT %MW21060.3 *) (* R366_1_M_O_RB_1_CYCLE_SET *)
    R366_1_M_O_RB_1차_작업완료_리셋 : BOOL; (* AT %MW21062.0 *) (* R366_1_M_O_RB_1차_작업완료_리셋 *)
    R366_1_M_O_RB_2차_작업완료_리셋 : BOOL; (* AT %MW21062.1 *) (* R366_1_M_O_RB_2차_작업완료_리셋 *)
    R366_1_M_O_RB_2차_진입OK : BOOL; (* AT %MW21061.8 *) (* R366_1_M_O_RB_2차_진입OK *)
    R366_1_M_O_RB_3차_작업완료_리셋 : BOOL; (* AT %MW21062.2 *) (* R366_1_M_O_RB_3차_작업완료_리셋 *)
    R366_1_M_O_RB_3차_진입OK : BOOL; (* AT %MW21061.9 *) (* R366_1_M_O_RB_3차_진입OK *)
    R366_1_M_O_RB_4차_작업완료_리셋 : BOOL; (* AT %MW21062.3 *) (* R366_1_M_O_RB_4차_작업완료_리셋 *)
    R366_1_M_O_RB_4차_진입OK : BOOL; (* AT %MW21061.10 *) (* R366_1_M_O_RB_4차_진입OK *)
    R366_1_M_O_RB_5차_작업완료_리셋 : BOOL; (* AT %MW21062.4 *) (* R366_1_M_O_RB_5차_작업완료_리셋 *)
    R366_1_M_O_RB_5차_진입OK : BOOL; (* AT %MW21061.11 *) (* R366_1_M_O_RB_5차_진입OK *)
    R366_1_M_O_RB_6차_작업완료_리셋 : BOOL; (* AT %MW21062.5 *) (* R366_1_M_O_RB_6차_작업완료_리셋 *)
    R366_1_M_O_RB_6차_진입OK : BOOL; (* AT %MW21061.12 *) (* R366_1_M_O_RB_6차_진입OK *)
    R366_1_M_O_RB_7차_작업완료_리셋 : BOOL; (* AT %MW21062.6 *) (* R366_1_M_O_RB_7차_작업완료_리셋 *)
    R366_1_M_O_RB_7차_진입OK : BOOL; (* AT %MW21061.13 *) (* R366_1_M_O_RB_7차_진입OK *)
    R366_1_M_O_RB_ATD_OK : BOOL; (* AT %MW21060.6 *) (* R366_1_M_O_RB_ATD_OK *)
    R366_1_M_O_RB_PLT_10_진입OK : BOOL; (* AT %MW21063.10 *) (* R366_1_M_O_RB_PLT_10_진입OK *)
    R366_1_M_O_RB_PLT_11_진입OK : BOOL; (* AT %MW21063.11 *) (* R366_1_M_O_RB_PLT_11_진입OK *)
    R366_1_M_O_RB_PLT_12_진입OK : BOOL; (* AT %MW21063.12 *) (* R366_1_M_O_RB_PLT_12_진입OK *)
    R366_1_M_O_RB_PLT_1_진입OK : BOOL; (* AT %MW21063.1 *) (* R366_1_M_O_RB_PLT_1_진입OK *)
    R366_1_M_O_RB_PLT_2_진입OK : BOOL; (* AT %MW21063.2 *) (* R366_1_M_O_RB_PLT_2_진입OK *)
    R366_1_M_O_RB_PLT_3_진입OK : BOOL; (* AT %MW21063.3 *) (* R366_1_M_O_RB_PLT_3_진입OK *)
    R366_1_M_O_RB_PLT_4_진입OK : BOOL; (* AT %MW21063.4 *) (* R366_1_M_O_RB_PLT_4_진입OK *)
    R366_1_M_O_RB_PLT_5_진입OK : BOOL; (* AT %MW21063.5 *) (* R366_1_M_O_RB_PLT_5_진입OK *)
    R366_1_M_O_RB_PLT_6_진입OK : BOOL; (* AT %MW21063.6 *) (* R366_1_M_O_RB_PLT_6_진입OK *)
    R366_1_M_O_RB_PLT_7_진입OK : BOOL; (* AT %MW21063.7 *) (* R366_1_M_O_RB_PLT_7_진입OK *)
    R366_1_M_O_RB_PLT_8_진입OK : BOOL; (* AT %MW21063.8 *) (* R366_1_M_O_RB_PLT_8_진입OK *)
    R366_1_M_O_RB_PLT_9_진입OK : BOOL; (* AT %MW21063.9 *) (* R366_1_M_O_RB_PLT_9_진입OK *)
    R366_1_M_O_RB_PLT_카운터리셋_보조 : BOOL; (* AT %MW21060.10 *) (* R366_1_M_O_RB_PLT_카운터리셋_보조 *)
    R366_1_M_O_RB_PROG_NO : WORD; (* AT %MW21064 *)
    R366_1_M_O_RB_RESTART_OK : BOOL; (* AT %MW21060.2 *) (* R366_1_M_O_RB_RESTART_OK *)
    R366_1_M_O_RB_START_OK : BOOL; (* AT %MW21060.0 *) (* R366_1_M_O_RB_START_OK *)
    R366_1_M_O_RB_TEST_MODE_5000회 : BOOL; (* AT %MW21060.12 *) (* R366_1_M_O_RB_TEST_MODE_5000회 *)
    R366_1_M_O_RB_TIP_교체_시작 : BOOL; (* AT %MW21060.7 *) (* R366_1_M_O_RB_TIP_교체_시작 *)
    R366_1_M_O_RB_TIP_교체_완료 : BOOL; (* AT %MW21060.8 *) (* R366_1_M_O_RB_TIP_교체_완료 *)
    R366_1_M_O_RB_VIP_MODE : BOOL; (* AT %MW21060.11 *) (* R366_1_M_O_RB_VIP_MODE *)
    R366_1_M_O_RB_냉각수_차단_요청 : BOOL; (* AT %MW21060.9 *) (* R366_1_M_O_RB_냉각수_차단_요청 *)
    R366_1_M_O_RB_진입OK_AX차종 : BOOL; (* AT %MW21061.0 *) (* R366_1_M_O_RB_진입OK_AX차종 *)
    R366_1_M_O_RB_진입OK_B차종 : BOOL; (* AT %MW21061.1 *) (* R366_1_M_O_RB_진입OK_B차종 *)
    R366_1_M_O_RB_진입OK_C차종 : BOOL; (* AT %MW21061.2 *) (* R366_1_M_O_RB_진입OK_C차종 *)
    R366_1_M_O_RB_진입OK_D차종 : BOOL; (* AT %MW21061.3 *) (* R366_1_M_O_RB_진입OK_D차종 *)
    R366_1_M_O_RB_진입OK_E차종 : BOOL; (* AT %MW21061.4 *) (* R366_1_M_O_RB_진입OK_E차종 *)
    R366_1_M_O_RB_진입OK_F차종 : BOOL; (* AT %MW21061.5 *) (* R366_1_M_O_RB_진입OK_F차종 *)
    R366_1_M_O_RB_진입OK_G차종 : BOOL; (* AT %MW21061.6 *) (* R366_1_M_O_RB_진입OK_G차종 *)
    R366_1_M_O_RB_진입OK_H차종 : BOOL; (* AT %MW21061.7 *) (* R366_1_M_O_RB_진입OK_H차종 *)
    R366_1_M_O_RB_최종_작업완료_리셋 : BOOL; (* AT %MW21060.5 *) (* R366_1_M_O_RB_최종_작업완료_리셋 *)
    R366_1_M_O_RB_프로그램_OK : BOOL; (* AT %MW21060.1 *) (* R366_1_M_O_RB_프로그램_OK *)
    R366_1_O_RB_OUTPUT : ARRAY[0..3] OF WORD; (* AT %MW94060 *) (* R366_1_O_RB_OUTPUT *)
    R369_1_M_I_RB_간섭무_1 : BOOL; (* AT %MW20082.0 *) (* R369_1_M_I_RB_간섭무_1 *)
END_VAR
(* ladder body could not be read *)
END_PROGRAM

PROGRAM S366_로보트_용접타점수 (* task: 스캔 프로그램 *)
VAR_EXTERNAL
    R364_1_I_RB_용접타점수 : WORD; (* AT %MW84055 *) (* R364_1_I_RB_용접타점수 *)
    R364_1_M_I_RB_1차_작업완료 : BOOL; (* AT %MW20051.2 *) (* R364_1_M_I_RB_1차_작업완료 *)
    R366_1_I_RB_용접타점수 : WORD; (* AT %MW84065 *) (* R366_1_I_RB_용접타점수 *)
END_VAR
VAR_EXTERNAL RETAIN
    R364_1_M_AX_차종_용접타점수 : WORD; (* AT %MW8010 *)
    R364_1_M_용접완료 : BOOL; (* AT %MW2006.1 *)
    R364_1_M_용접타점수_OK : BOOL; (* AT %MW2006.8 *)
    R366_1_M_용접완료 : BOOL; (* AT %MW3006.1 *)
    R366_1_M_용접타점수_OK : BOOL; (* AT %MW3006.8 *)
    S364_M_전체_용접완료 : BOOL; (* AT %MW2006.0 *)
    S366_M_R366_1_용접완료 : BOOL; (* AT %MW3001.3 *)
    S366_M_전체_용접완료 : BOOL; (* AT %MW3006.0 *)
    S366_M_차종1_AX : BOOL; (* AT %MW10161.0 *) (* S366 M 차종1 AX *)
END_VAR
VAR
    _t1 : BOOL;
END_VAR

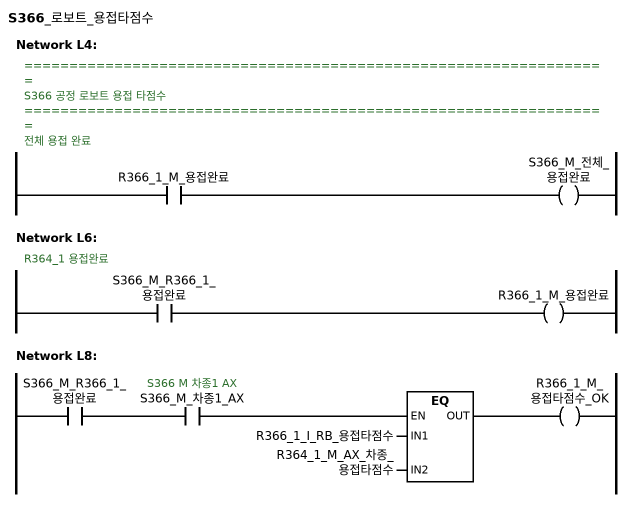
(* ================================================================= *)
(* S366 공정 로보트 용접 타점수 *)
(* ================================================================= *)
(* 전체 용접 완료 *)
(* Rung L4 *)
S366_M_전체_용접완료 := R366_1_M_용접완료;
(* R364_1 용접완료 *)
(* Rung L6 *)
R366_1_M_용접완료 := S366_M_R366_1_용접완료;
(* Rung L8 *)
IF S366_M_R366_1_용접완료 AND S366_M_차종1_AX THEN _t1 := R366_1_I_RB_용접타점수 = R364_1_M_AX_차종_용접타점수; END_IF;
R366_1_M_용접타점수_OK := _t1;
END_PROGRAM

PROGRAM S366_이상 (* task: 스캔 프로그램 *)
VAR
    INST : TON;
    INST1 : TON;
    INST10 : TON;
    INST11 : TON;
    INST12 : TON;
    INST13 : TON;
    INST14 : TON;
    INST15 : TON;
    INST16 : TON;
    INST17 : TON;
    INST18 : TON;
    INST19 : TON;
    INST2 : TON;
    INST20 : TON;
    INST21 : TON;
    INST22 : TON;
    INST23 : TON;
    INST24 : TON;
    INST25 : TON;
    INST26 : TON;
    INST27 : TON;
    INST28 : TON;
    INST29 : TON;
    INST3 : TON;
    INST30 : TON;
    INST31 : TON;
    INST32 : TON;
    INST33 : TON;
    INST34 : TON;
    INST35 : TON;
    INST36 : TON;
    INST37 : TON;
    INST38 : TON;
    INST39 : TON;
    INST4 : TON;
    INST40 : TON;
    INST41 : TON;
    INST42 : TON;
    INST43 : TON;
    INST5 : TON;
    INST6 : TON;
    INST7 : TON;
    INST8 : TON;
    INST9 : TON;
    T366_LH_TURN_LS_이상 : TON;
    T366_RH_TURN_LS_이상 : TON;
END_VAR
VAR_EXTERNAL
    R361_1_M_I_RB_이상 : BOOL; (* AT %MW20010.2 *) (* R361_1_M_I_RB_이상 *)
    R361_1_M_I_RB_프로그램_이상 : BOOL; (* AT %MW20010.6 *) (* R361_1_M_I_RB_프로그램_이상 *)
    R366_1_M_I_RB_이상 : BOOL; (* AT %MW20060.2 *) (* R366_1_M_I_RB_이상 *)
    R366_1_M_I_RB_프로그램_이상 : BOOL; (* AT %MW20060.6 *) (* R366_1_M_I_RB_프로그램_이상 *)
    S362_6_INV1_NFB_ON : BOOL; (* AT %MW85013.0 *) (* S362_6_INV1_NFB_ON *)
    S362_6_INV1_NOMAL_OK : BOOL; (* AT %MW85010.0 *) (* S362_6_INV1_NOMAL_OK *)
    S362_6_INV3_BRAKE_CR_ON : BOOL; (* AT %MW95015.7 *) (* S362_6_INV3_BRAKE_CR_ON *)
    S362_6_INV3_MC_BRAKE_ON : BOOL; (* AT %MW85010.9 *) (* S362_6_INV3_MC_BRAKE_ON *)
    S362_6_INV3_NFB_ON : BOOL; (* AT %MW85013.2 *) (* S362_6_INV3_NFB_ON *)
    S362_6_INV3_NOMAL_OK : BOOL; (* AT %MW85010.8 *) (* S362_6_INV3_NOMAL_OK *)
    S362_6_INV3_RETURN : BOOL; (* AT %MW95015.1 *) (* S362_6_INV3_RETURN *)
    S362_6_INV3_TURN : BOOL; (* AT %MW95015.0 *) (* S362_6_INV3_TURN *)
    S362_6_INV4_BRAKE_CR_ON : BOOL; (* AT %MW95015.15 *) (* S362_6_INV4_BRAKE_CR_ON *)
    S362_6_INV4_MC_BRAKE_ON : BOOL; (* AT %MW85010.13 *) (* S362_6_INV4_MC_BRAKE_ON *)
    S362_6_INV4_NFB_ON : BOOL; (* AT %MW85013.3 *) (* S362_6_INV4_NFB_ON *)
    S362_6_INV4_NOMAL_OK : BOOL; (* AT %MW85010.12 *) (* S362_6_INV4_NOMAL_OK *)
    S362_6_INV4_RETURN : BOOL; (* AT %MW95015.9 *) (* S362_6_INV4_RETURN *)
    S362_6_INV4_TURN : BOOL; (* AT %MW95015.8 *) (* S362_6_INV4_TURN *)
    S366R_8_10_PLC_BOX_CP_TRIP : BOOL; (* AT %MW88100.15 *) (* S366L_LS_AX_MAINTENANCE_CHK *)
    S366R_8_20_PLC_BOX_CP_TRIP : BOOL; (* AT %MW88200.15 *) (* S366R_LS_AX_MAINTENANCE_CHK *)
    S366_6_10_PLC_BOX_CP_TRIP : BOOL; (* AT %MW86102.15 *) (* S366_6_10_PLC_BOX_CP_TRIP *)
    S366_INDEX_LH_TURN_감지1 : BOOL; (* AT %MW86101.4 *) (* S366_INDEX_LH_TURN_감지1 *)
    S366_INDEX_LH_TURN_감지2 : BOOL; (* AT %MW86101.5 *) (* S366_INDEX_LH_TURN_감지2 *)
    S366_INDEX_LH_TURN_감지3 : BOOL; (* AT %MW86101.6 *) (* S366_INDEX_LH_TURN_감지3 *)
    S366_INDEX_LH_TURN_원점 : BOOL; (* AT %MW86101.7 *) (* S366_INDEX_LH_TURN_원점 *)
    S366_INDEX_RH_TURN_감지1 : BOOL; (* AT %MW86101.0 *) (* S366_INDEX_RH_TURN_감지1 *)
    S366_INDEX_RH_TURN_감지2 : BOOL; (* AT %MW86101.1 *) (* S366_INDEX_RH_TURN_감지2 *)
    S366_INDEX_RH_TURN_감지3 : BOOL; (* AT %MW86101.2 *) (* S366_INDEX_RH_TURN_감지3 *)
    S366_INDEX_RH_TURN_원점 : BOOL; (* AT %MW86101.3 *) (* S366_INDEX_RH_TURN_원점 *)
    S366_LH_CUT_OFF_BOX_ON : BOOL; (* AT %MW86102.10 *)
    S366_RH_CUT_OFF_BOX_ON : BOOL; (* AT %MW86102.11 *)
    S366_공기압_AIR_CHECK : BOOL; (* AT %MW86102.14 *) (* S366_공기압_AIR_CHECK *)
    _0004_EB05_CFG_ER : BOOL; (* AT %MW184032.0 *) (* EB 구성 에러 *)
    _0004_EB05_DEER : BOOL; (* AT %MW184032.1 *) (* EB 운전 중 탈락 *)
    _0004_EB06_CFG_ER : BOOL; (* AT %MW184034.8 *) (* EB 구성 에러 *)
    _0004_EB06_DEER : BOOL; (* AT %MW184034.9 *) (* EB 운전 중 탈락 *)
    _0006_EB10_CFG_ER : BOOL; (* AT %MW186028.0 *) (* EB 구성 에러 *)
    _0006_EB10_DEER : BOOL; (* AT %MW186028.1 *) (* EB 운전 중 탈락 *)
    _0006_EB10_IO_DEER : BOOL; (* AT %MW186029.2 *) (* EB IO 탈락 에러 *)
    _0006_EB10_IO_TYER : BOOL; (* AT %MW186029.1 *) (* EB IO 타입 에러 *)
    _0006_EB41_CFG_ER : BOOL; (* AT %MW186064.0 *) (* EB 구성 에러 *)
    _0006_EB41_DEER : BOOL; (* AT %MW186064.1 *) (* EB 운전 중 탈락 *)
    _0006_EB41_IO_DEER : BOOL; (* AT %MW186065.2 *) (* EB IO 탈락 에러 *)
    _0006_EB41_IO_TYER : BOOL; (* AT %MW186065.1 *) (* EB IO 타입 에러 *)
END_VAR
VAR_EXTERNAL RETAIN
    R366_1_M_NODE_4_06_통신_이상 : BOOL; (* AT %MW3024.8 *)
    R366_1_M_용접_카운트_이상 : BOOL; (* AT %MW3029.0 *)
    R366_1_M_용접타점수_OK : BOOL; (* AT %MW3006.8 *)
    S362_M_공정_불간섭 : BOOL; (* AT %MW1004.1 *) (* S362_M_공정_불간섭 *)
    S362_M_공정_제품감지_무 : BOOL; (* AT %MW1001.5 *) (* S362_M_공정_제품감지_무 *)
    S362_M_공정_차종_유 : BOOL; (* AT %MW1002.0 *) (* S362_M_공정_차종_유 *)
    S362_M_자동_운전중 : BOOL; (* AT %MW1000.4 *) (* S362 자동운전중 *)
    S366_LH_M_NODE_8_10_통신_이상 : BOOL; (* AT %MW3024.1 *)
    S366_M_AX_LH_CLP_전진_LS_이상 : BOOL; (* AT %MW3104.5 *) (* S366_M_AX_LH_CLP_전진_LS_이상 *)
    S366_M_AX_LH_CLP_후진_LS_이상 : BOOL; (* AT %MW3104.6 *) (* S366_M_AX_LH_CLP_후진_LS_이상 *)
    S366_M_AX_RH_CLP_전진_LS_이상 : BOOL; (* AT %MW3112.5 *) (* S366_M_AX_RH_CLP_전진_LS_이상 *)
    S366_M_AX_RH_CLP_후진_LS_이상 : BOOL; (* AT %MW3112.6 *) (* S366_M_AX_RH_CLP_후진_LS_이상 *)
    S366_M_CP_OFF : BOOL; (* AT %MW3017.0 *)
    S366_M_LH_CB_OFF : BOOL; (* AT %MW3021.2 *)
    S366_M_LH_CP_OFF : BOOL; (* AT %MW3017.2 *) (* S366_M_LH_CP_OFF *)
    S366_M_LH_INV_이상 : BOOL; (* AT %MW3019.0 *) (* S366_M_LH_INV_이상 *)
    S366_M_LH_MC_이상 : BOOL; (* AT %MW3023.0 *) (* S366_M_LH_MC_이상 *)
    S366_M_LH_NFB_OFF : BOOL; (* AT %MW3021.0 *) (* S366_M_LH_NFB_OFF *)
    S366_M_LH_TURN_1_포지션단 : BOOL; (* AT %MW3101.3 *) (* S366_M_LH_TURN_1_포지션단 *)
    S366_M_LH_TURN_2_포지션단 : BOOL; (* AT %MW3101.4 *) (* S366_M_LH_TURN_2_포지션단 *)
    S366_M_LH_TURN_3_포지션단 : BOOL; (* AT %MW3101.5 *) (* S366_M_LH_TURN_3_포지션단 *)
    S366_M_LH_TURN_4_포지션단 : BOOL; (* AT %MW3101.6 *) (* S366_M_LH_TURN_4_포지션단 *)
    S366_M_LH_TURN_LS_이상 : BOOL; (* AT %MW3101.7 *) (* S366_M_LH_TURN_LS_이상 *)
    S366_M_LH_TURN_조건 : BOOL; (* AT %MW3101.0 *) (* S366_M_LH_TURN_조건 *)
    S366_M_NODE_6_10_통신_이상 : BOOL; (* AT %MW3024.0 *)
    S366_M_R361_1_ROOF_로딩완료 : BOOL; (* AT %MW3001.2 *)
    S366_M_R361_1_동일차종_OK : BOOL; (* AT %MW3005.8 *)
    S366_M_R361_1_차종매칭_조건 : BOOL; (* AT %MW3005.0 *)
    S366_M_R363_2_RAIL_로딩완료 : BOOL; (* AT %MW3001.1 *)
    S366_M_R366_1_용접완료 : BOOL; (* AT %MW3001.3 *)
    S366_M_RH_CB_OFF : BOOL; (* AT %MW3021.3 *)
    S366_M_RH_CP_OFF : BOOL; (* AT %MW3017.3 *) (* S366_M_RH_CP_OFF *)
    S366_M_RH_INV_이상 : BOOL; (* AT %MW3019.1 *) (* S366_M_RH_INV_이상 *)
    S366_M_RH_MC_이상 : BOOL; (* AT %MW3023.1 *) (* S366_M_RH_MC_이상 *)
    S366_M_RH_NFB_OFF : BOOL; (* AT %MW3021.1 *) (* S366_M_RH_NFB_OFF *)
    S366_M_RH_TURN_1_포지션단 : BOOL; (* AT %MW3109.3 *) (* S366_M_RH_TURN_1_포지션단 *)
    S366_M_RH_TURN_2_포지션단 : BOOL; (* AT %MW3109.4 *) (* S366_M_RH_TURN_2_포지션단 *)
    S366_M_RH_TURN_3_포지션단 : BOOL; (* AT %MW3109.5 *) (* S366_M_RH_TURN_3_포지션단 *)
    S366_M_RH_TURN_4_포지션단 : BOOL; (* AT %MW3109.6 *) (* S366_M_RH_TURN_4_포지션단 *)
    S366_M_RH_TURN_LS_이상 : BOOL; (* AT %MW3109.7 *) (* S366_M_RH_TURN_LS_이상 *)
    S366_M_RH_TURN_조건 : BOOL; (* AT %MW3109.0 *) (* S366_M_RH_TURN_조건 *)
    S366_M_SAFETY_불간섭 : BOOL; (* AT %MW3004.4 *) (* S366_M_SAFETY_불간섭 *)
    S366_M_TURN_LOCK_전진_LS_이상 : BOOL; (* AT %MW3100.5 *) (* S366_M_TURN_LOCK_전진_LS_이상 *)
    S366_M_TURN_LOCK_후진_LS_이상 : BOOL; (* AT %MW3100.6 *) (* S366_M_TURN_LOCK_후진_LS_이상 *)
    S366_M_공정_AX_FRT_PNL_제품감지_이상 : BOOL; (* AT %MW3014.4 *)
    S366_M_공정_AX_RAIL_제품감지_이상 : BOOL; (* AT %MW3014.3 *)
    S366_M_공정_AX_RR_PNL_제품감지_이상 : BOOL; (* AT %MW3014.5 *)
    S366_M_공정_AX_공용_제품감지_이상 : BOOL; (* AT %MW3014.0 *)
    S366_M_공정_AX_썬루프_제품감지_이상 : BOOL; (* AT %MW3014.2 *)
    S366_M_공정_AX_일반루프_제품감지_이상 : BOOL; (* AT %MW3014.1 *)
    S366_M_공정_FRT_PNL_제품감지_유 : BOOL; (* AT %MW3002.12 *)
    S366_M_공정_RAIL_제품감지_유 : BOOL; (* AT %MW3001.14 *)
    S366_M_공정_RR_PNL_제품감지_유 : BOOL; (* AT %MW3002.14 *)
    S366_M_공정_공용_제품감지_유 : BOOL; (* AT %MW3001.8 *)
    S366_M_공정_불간섭 : BOOL; (* AT %MW3004.1 *) (* S366_M_공정_불간섭 *)
    S366_M_공정_썬루프_제품감지_유 : BOOL; (* AT %MW3001.12 *)
    S366_M_공정_일반루프_제품감지_유 : BOOL; (* AT %MW3001.10 *)
    S366_M_공정_제품감지_무 : BOOL; (* AT %MW3001.7 *) (* S366_M_공정_제품감지_무 *)
    S366_M_공정_차종_유 : BOOL; (* AT %MW3002.0 *) (* S366_M_공정_차종_유 *)
    S366_M_썬루프_사양_이상 : BOOL; (* AT %MW3016.1 *)
    S366_M_일반루프_사양_이상 : BOOL; (* AT %MW3016.0 *)
    S366_M_자동_운전중 : BOOL; (* AT %MW3000.4 *) (* S366 자동운전중 *)
    S366_M_차종6_썬루프 : BOOL; (* AT %MW10163.4 *) (* S366 M 차종6 썬루프 *)
    S366_M_차종6_일반루프 : BOOL; (* AT %MW10163.3 *) (* S366 M 차종6 일반루프 *)
    S366_M_총괄_CP_이상 : BOOL; (* AT %MW3009.7 *) (* S366 CP OFF 이상 *)
    S366_M_총괄_CT_이상 : BOOL; (* AT %MW3010.4 *) (* S366   TACK TIME 이상 *)
    S366_M_총괄_EOCR_이상 : BOOL; (* AT %MW3009.8 *) (* S366_M_총괄_EOCR_이상 *)
    S366_M_총괄_INV_이상 : BOOL; (* AT %MW3009.9 *) (* S366 인버터 이상 *)
    S366_M_총괄_LS_이상 : BOOL; (* AT %MW3009.15 *) (* S366 LS 이상 *)
    S366_M_총괄_MATCH_이상 : BOOL; (* AT %MW3010.0 *) (* S366 매트SW 이상 *)
    S366_M_총괄_MC_이상 : BOOL; (* AT %MW3009.13 *) (* S366 MC 이상 *)
    S366_M_총괄_NFB_이상 : BOOL; (* AT %MW3009.11 *) (* S366 NFB 이상 *)
    S366_M_총괄_ROBOT_이상 : BOOL; (* AT %MW3010.1 *) (* S366 ROBOT 이상 *)
    S366_M_총괄_SAFETY_이상 : BOOL; (* AT %MW3009.2 *) (* S366_M_총괄_SAFETY_이상 *)
    S366_M_총괄_공기압_이상 : BOOL; (* AT %MW3009.3 *) (* S366 공기압 이상 *)
    S366_M_총괄_사양_이상 : BOOL; (* AT %MW3009.6 *) (* S366 사양 이상 *)
    S366_M_총괄_오버런_이상 : BOOL; (* AT %MW3009.12 *) (* S366 OVER RUN 이상 *)
    S366_M_총괄_용접타점수_이상 : BOOL; (* AT %MW3010.2 *) (* S366 용접타점수 이상 *)
    S366_M_총괄_이상 : BOOL; (* AT %MW3009.0 *) (* S366_M_총괄_이상 *)
    S366_M_총괄_제품감지_이상 : BOOL; (* AT %MW3009.4 *) (* S366 제품감지 이상 *)
    S366_M_총괄_차종_이상 : BOOL; (* AT %MW3009.5 *) (* S366 차종 이상 *)
    S366_M_총괄_통신_이상 : BOOL; (* AT %MW3009.14 *) (* S366 통신이상 *)
    S366_RH_M_NODE_8_20_통신_이상 : BOOL; (* AT %MW3024.2 *)
    전체_M_이상_리셋 : BOOL; (* AT %MW308.2 *) (* ALL공정 PB 이상리셋 *)
END_VAR

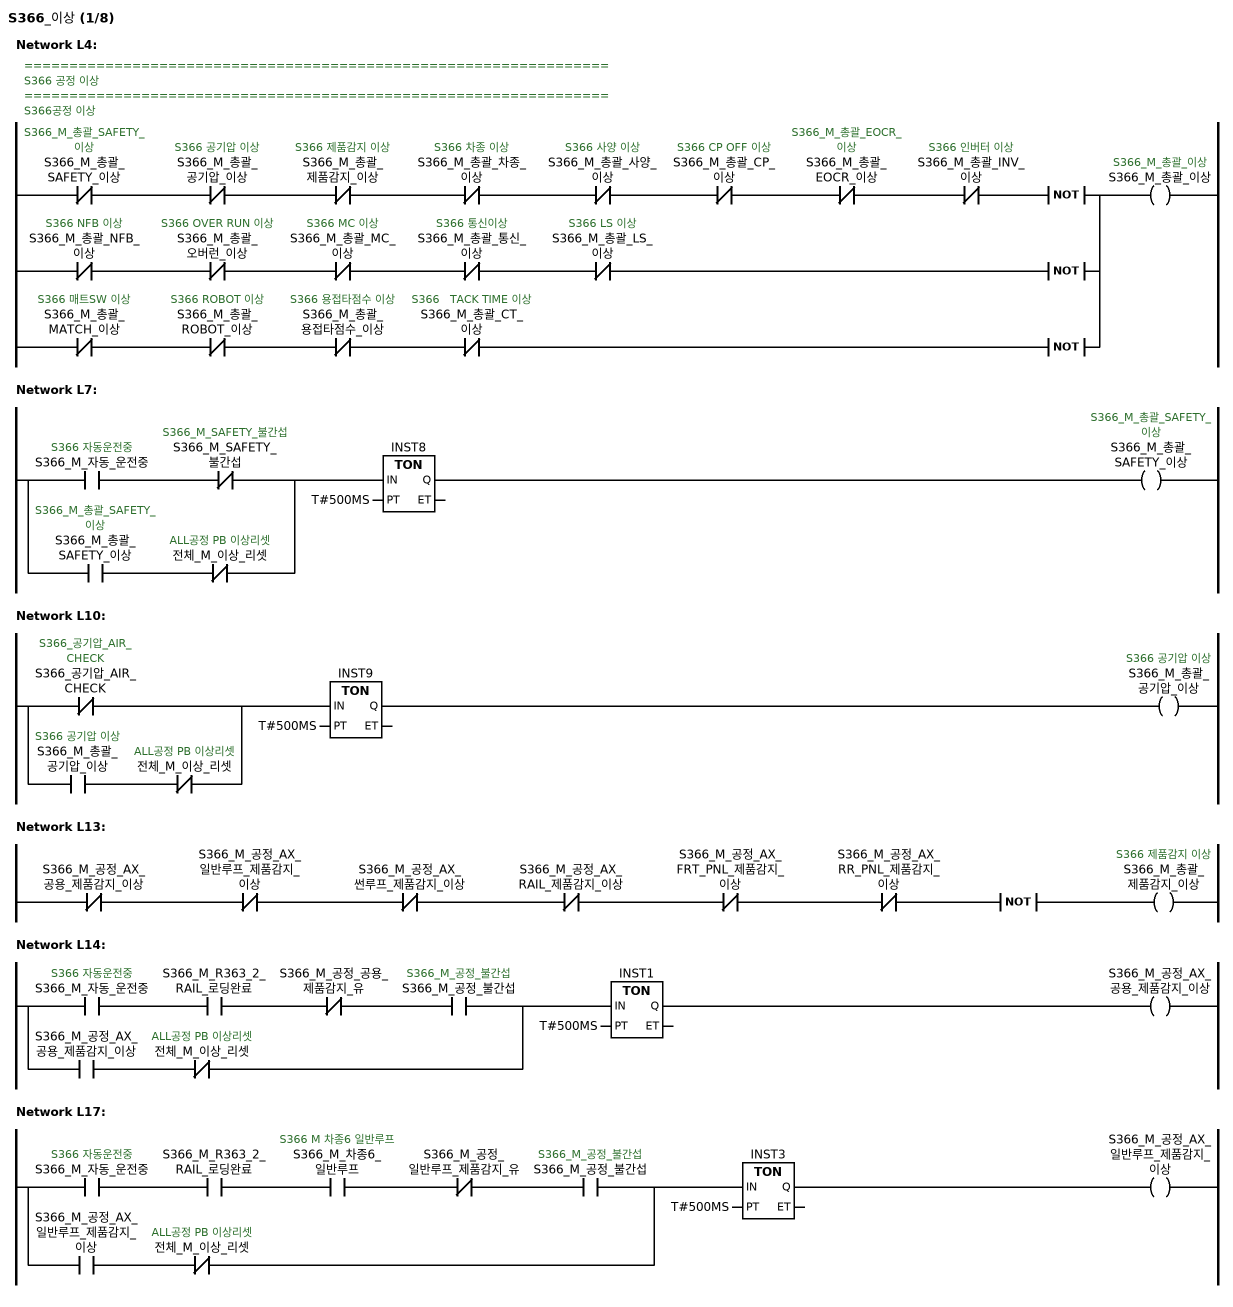
(* ================================================================= *)
(* S366 공정 이상 *)
(* ================================================================= *)
(* S366공정 이상 *)
(* Rung L4 *)
S366_M_총괄_이상 := NOT (NOT S366_M_총괄_SAFETY_이상 AND NOT S366_M_총괄_공기압_이상 AND NOT S366_M_총괄_제품감지_이상 AND NOT S366_M_총괄_차종_이상 AND NOT S366_M_총괄_사양_이상 AND NOT S366_M_총괄_CP_이상 AND NOT S366_M_총괄_EOCR_이상 AND NOT S366_M_총괄_INV_이상) OR NOT (NOT S366_M_총괄_NFB_이상 AND NOT S366_M_총괄_오버런_이상 AND NOT S366_M_총괄_MC_이상 AND NOT S366_M_총괄_통신_이상 AND NOT S366_M_총괄_LS_이상) OR NOT (NOT S366_M_총괄_MATCH_이상 AND NOT S366_M_총괄_ROBOT_이상 AND NOT S366_M_총괄_용접타점수_이상 AND NOT S366_M_총괄_CT_이상);
(* Rung L7 *)
INST8(IN := (S366_M_자동_운전중 AND NOT S366_M_SAFETY_불간섭) OR (S366_M_총괄_SAFETY_이상 AND NOT 전체_M_이상_리셋), PT := T#500MS);
S366_M_총괄_SAFETY_이상 := INST8.Q;
(* Rung L10 *)
INST9(IN := NOT S366_공기압_AIR_CHECK OR (S366_M_총괄_공기압_이상 AND NOT 전체_M_이상_리셋), PT := T#500MS);
S366_M_총괄_공기압_이상 := INST9.Q;
(* Rung L13 *)
S366_M_총괄_제품감지_이상 := NOT (NOT S366_M_공정_AX_공용_제품감지_이상 AND NOT S366_M_공정_AX_일반루프_제품감지_이상 AND NOT S366_M_공정_AX_썬루프_제품감지_이상 AND NOT S366_M_공정_AX_RAIL_제품감지_이상 AND NOT S366_M_공정_AX_FRT_PNL_제품감지_이상 AND NOT S366_M_공정_AX_RR_PNL_제품감지_이상);
(* Rung L14 *)
INST1(IN := (S366_M_자동_운전중 AND S366_M_R363_2_RAIL_로딩완료 AND NOT S366_M_공정_공용_제품감지_유 AND S366_M_공정_불간섭) OR (S366_M_공정_AX_공용_제품감지_이상 AND NOT 전체_M_이상_리셋), PT := T#500MS);
S366_M_공정_AX_공용_제품감지_이상 := INST1.Q;
(* Rung L17 *)
INST3(IN := (S366_M_자동_운전중 AND S366_M_R363_2_RAIL_로딩완료 AND S366_M_차종6_일반루프 AND NOT S366_M_공정_일반루프_제품감지_유 AND S366_M_공정_불간섭) OR (S366_M_공정_AX_일반루프_제품감지_이상 AND NOT 전체_M_이상_리셋), PT := T#500MS);
S366_M_공정_AX_일반루프_제품감지_이상 := INST3.Q;

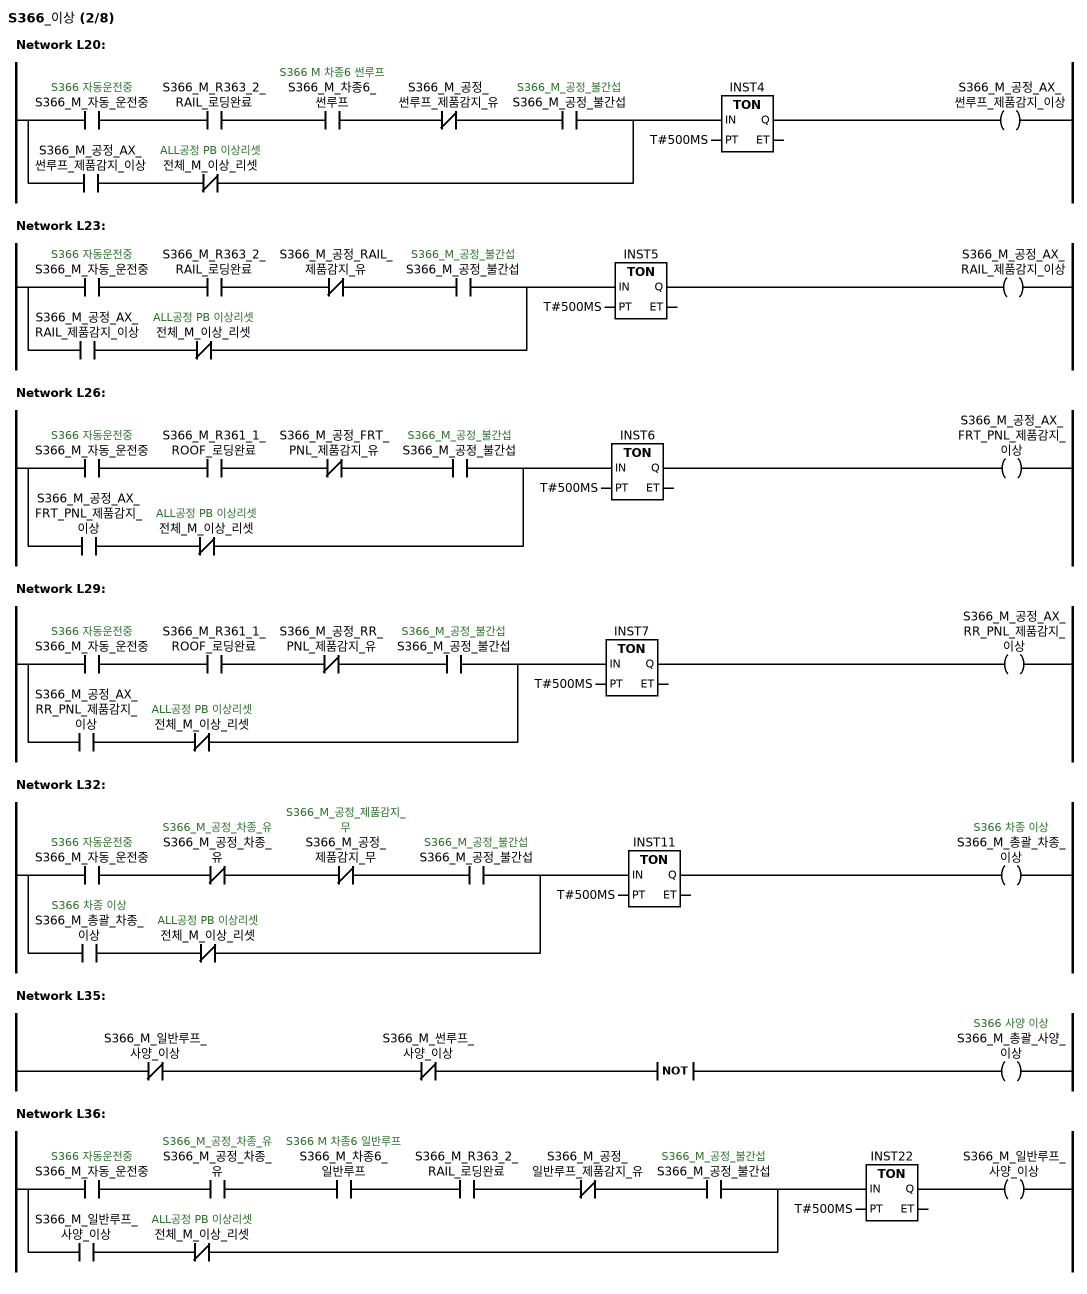
(* Rung L20 *)
INST4(IN := (S366_M_자동_운전중 AND S366_M_R363_2_RAIL_로딩완료 AND S366_M_차종6_썬루프 AND NOT S366_M_공정_썬루프_제품감지_유 AND S366_M_공정_불간섭) OR (S366_M_공정_AX_썬루프_제품감지_이상 AND NOT 전체_M_이상_리셋), PT := T#500MS);
S366_M_공정_AX_썬루프_제품감지_이상 := INST4.Q;
(* Rung L23 *)
INST5(IN := (S366_M_자동_운전중 AND S366_M_R363_2_RAIL_로딩완료 AND NOT S366_M_공정_RAIL_제품감지_유 AND S366_M_공정_불간섭) OR (S366_M_공정_AX_RAIL_제품감지_이상 AND NOT 전체_M_이상_리셋), PT := T#500MS);
S366_M_공정_AX_RAIL_제품감지_이상 := INST5.Q;
(* Rung L26 *)
INST6(IN := (S366_M_자동_운전중 AND S366_M_R361_1_ROOF_로딩완료 AND NOT S366_M_공정_FRT_PNL_제품감지_유 AND S366_M_공정_불간섭) OR (S366_M_공정_AX_FRT_PNL_제품감지_이상 AND NOT 전체_M_이상_리셋), PT := T#500MS);
S366_M_공정_AX_FRT_PNL_제품감지_이상 := INST6.Q;
(* Rung L29 *)
INST7(IN := (S366_M_자동_운전중 AND S366_M_R361_1_ROOF_로딩완료 AND NOT S366_M_공정_RR_PNL_제품감지_유 AND S366_M_공정_불간섭) OR (S366_M_공정_AX_RR_PNL_제품감지_이상 AND NOT 전체_M_이상_리셋), PT := T#500MS);
S366_M_공정_AX_RR_PNL_제품감지_이상 := INST7.Q;
(* Rung L32 *)
INST11(IN := (S366_M_자동_운전중 AND NOT S366_M_공정_차종_유 AND NOT S366_M_공정_제품감지_무 AND S366_M_공정_불간섭) OR (S366_M_총괄_차종_이상 AND NOT 전체_M_이상_리셋), PT := T#500MS);
S366_M_총괄_차종_이상 := INST11.Q;
(* Rung L35 *)
S366_M_총괄_사양_이상 := NOT (NOT S366_M_일반루프_사양_이상 AND NOT S366_M_썬루프_사양_이상);
(* Rung L36 *)
INST22(IN := (S366_M_자동_운전중 AND S366_M_공정_차종_유 AND S366_M_차종6_일반루프 AND S366_M_R363_2_RAIL_로딩완료 AND NOT S366_M_공정_일반루프_제품감지_유 AND S366_M_공정_불간섭) OR (S366_M_일반루프_사양_이상 AND NOT 전체_M_이상_리셋), PT := T#500MS);
S366_M_일반루프_사양_이상 := INST22.Q;

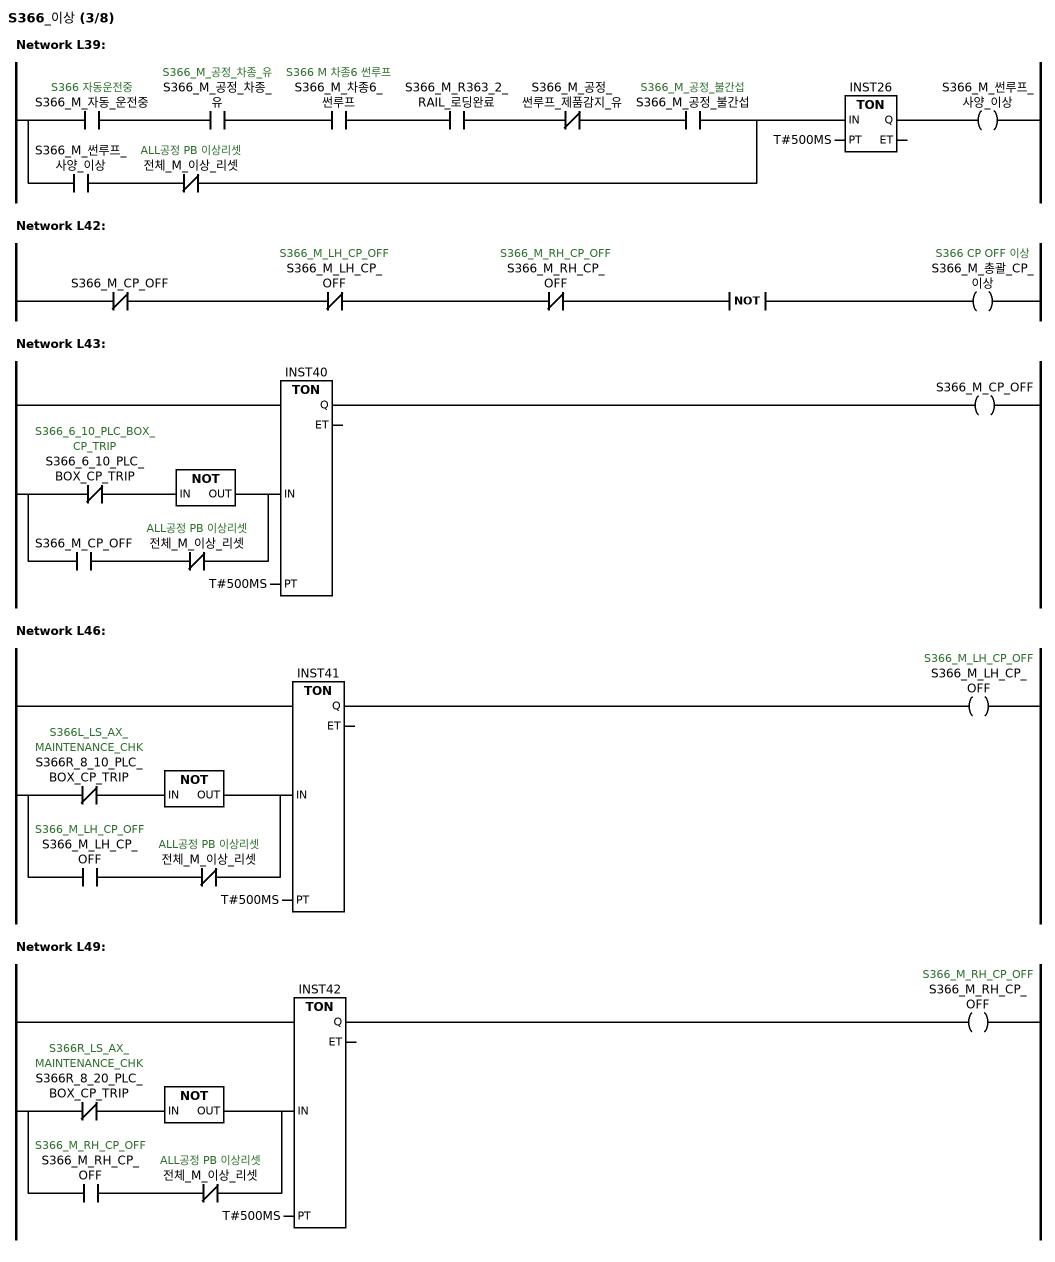
(* Rung L39 *)
INST26(IN := (S366_M_자동_운전중 AND S366_M_공정_차종_유 AND S366_M_차종6_썬루프 AND S366_M_R363_2_RAIL_로딩완료 AND NOT S366_M_공정_썬루프_제품감지_유 AND S366_M_공정_불간섭) OR (S366_M_썬루프_사양_이상 AND NOT 전체_M_이상_리셋), PT := T#500MS);
S366_M_썬루프_사양_이상 := INST26.Q;
(* Rung L42 *)
S366_M_총괄_CP_이상 := NOT (NOT S366_M_CP_OFF AND NOT S366_M_LH_CP_OFF AND NOT S366_M_RH_CP_OFF);
(* Rung L43 *)
INST40(IN := (NOT (NOT S366_6_10_PLC_BOX_CP_TRIP)) OR (S366_M_CP_OFF AND NOT 전체_M_이상_리셋), PT := T#500MS);
S366_M_CP_OFF := INST40.Q;
(* Rung L46 *)
INST41(IN := (NOT (NOT S366R_8_10_PLC_BOX_CP_TRIP)) OR (S366_M_LH_CP_OFF AND NOT 전체_M_이상_리셋), PT := T#500MS);
S366_M_LH_CP_OFF := INST41.Q;
(* Rung L49 *)
INST42(IN := (NOT (NOT S366R_8_20_PLC_BOX_CP_TRIP)) OR (S366_M_RH_CP_OFF AND NOT 전체_M_이상_리셋), PT := T#500MS);
S366_M_RH_CP_OFF := INST42.Q;

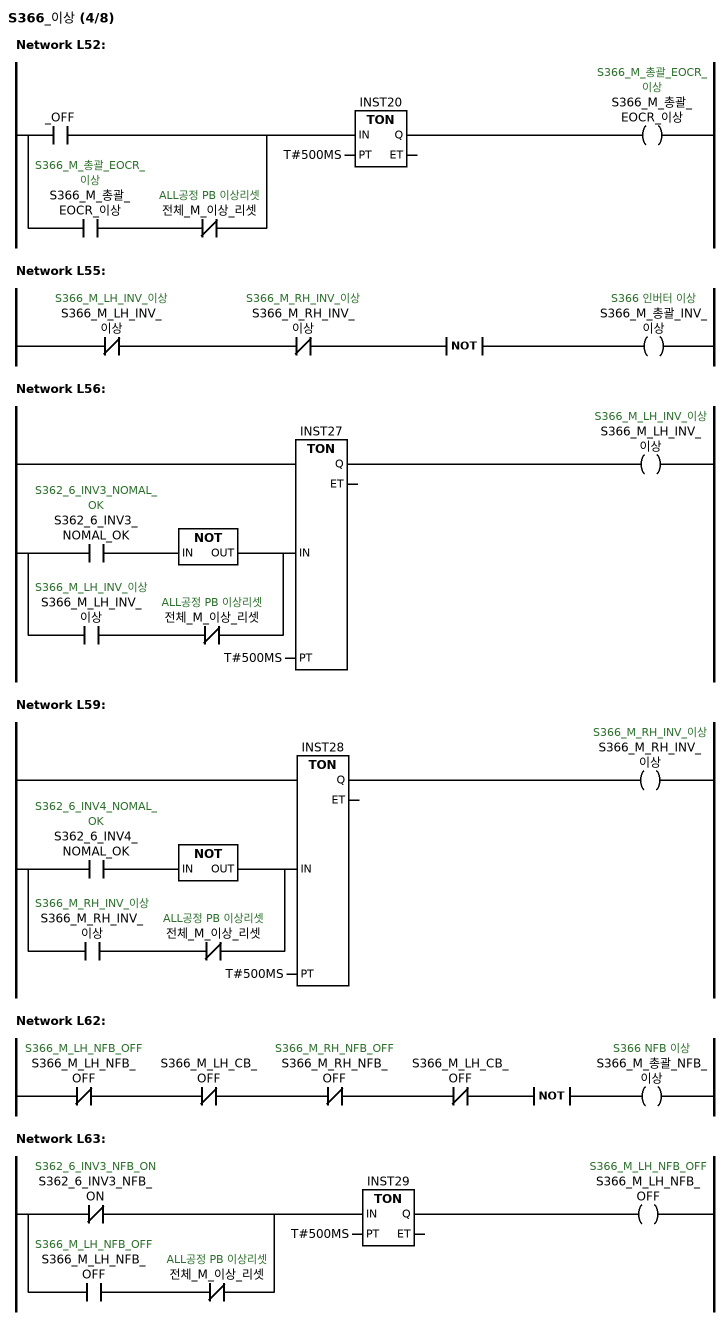
(* Rung L52 *)
INST20(IN := _OFF OR (S366_M_총괄_EOCR_이상 AND NOT 전체_M_이상_리셋), PT := T#500MS);
S366_M_총괄_EOCR_이상 := INST20.Q;
(* Rung L55 *)
S366_M_총괄_INV_이상 := NOT (NOT S366_M_LH_INV_이상 AND NOT S366_M_RH_INV_이상);
(* Rung L56 *)
INST27(IN := (NOT S362_6_INV3_NOMAL_OK) OR (S366_M_LH_INV_이상 AND NOT 전체_M_이상_리셋), PT := T#500MS);
S366_M_LH_INV_이상 := INST27.Q;
(* Rung L59 *)
INST28(IN := (NOT S362_6_INV4_NOMAL_OK) OR (S366_M_RH_INV_이상 AND NOT 전체_M_이상_리셋), PT := T#500MS);
S366_M_RH_INV_이상 := INST28.Q;
(* Rung L62 *)
S366_M_총괄_NFB_이상 := NOT (NOT S366_M_LH_NFB_OFF AND NOT S366_M_LH_CB_OFF AND NOT S366_M_RH_NFB_OFF AND NOT S366_M_LH_CB_OFF);
(* Rung L63 *)
INST29(IN := NOT S362_6_INV3_NFB_ON OR (S366_M_LH_NFB_OFF AND NOT 전체_M_이상_리셋), PT := T#500MS);
S366_M_LH_NFB_OFF := INST29.Q;

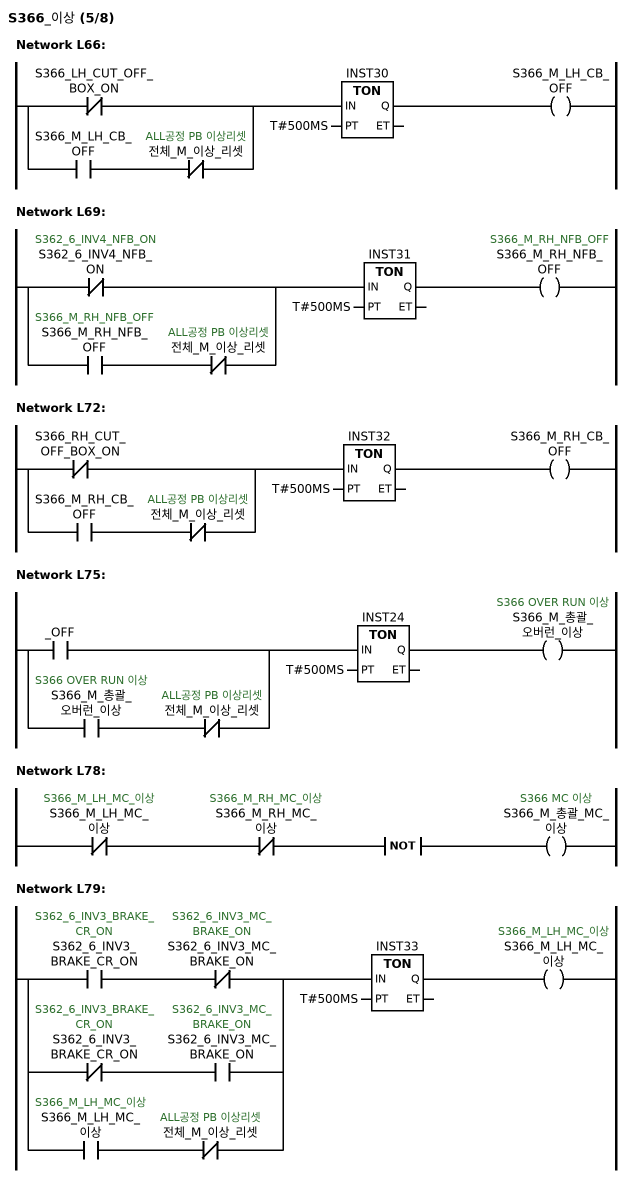
(* Rung L66 *)
INST30(IN := NOT S366_LH_CUT_OFF_BOX_ON OR (S366_M_LH_CB_OFF AND NOT 전체_M_이상_리셋), PT := T#500MS);
S366_M_LH_CB_OFF := INST30.Q;
(* Rung L69 *)
INST31(IN := NOT S362_6_INV4_NFB_ON OR (S366_M_RH_NFB_OFF AND NOT 전체_M_이상_리셋), PT := T#500MS);
S366_M_RH_NFB_OFF := INST31.Q;
(* Rung L72 *)
INST32(IN := NOT S366_RH_CUT_OFF_BOX_ON OR (S366_M_RH_CB_OFF AND NOT 전체_M_이상_리셋), PT := T#500MS);
S366_M_RH_CB_OFF := INST32.Q;
(* Rung L75 *)
INST24(IN := _OFF OR (S366_M_총괄_오버런_이상 AND NOT 전체_M_이상_리셋), PT := T#500MS);
S366_M_총괄_오버런_이상 := INST24.Q;
(* Rung L78 *)
S366_M_총괄_MC_이상 := NOT (NOT S366_M_LH_MC_이상 AND NOT S366_M_RH_MC_이상);
(* Rung L79 *)
INST33(IN := (S362_6_INV3_BRAKE_CR_ON AND NOT S362_6_INV3_MC_BRAKE_ON) OR (NOT S362_6_INV3_BRAKE_CR_ON AND S362_6_INV3_MC_BRAKE_ON) OR (S366_M_LH_MC_이상 AND NOT 전체_M_이상_리셋), PT := T#500MS);
S366_M_LH_MC_이상 := INST33.Q;

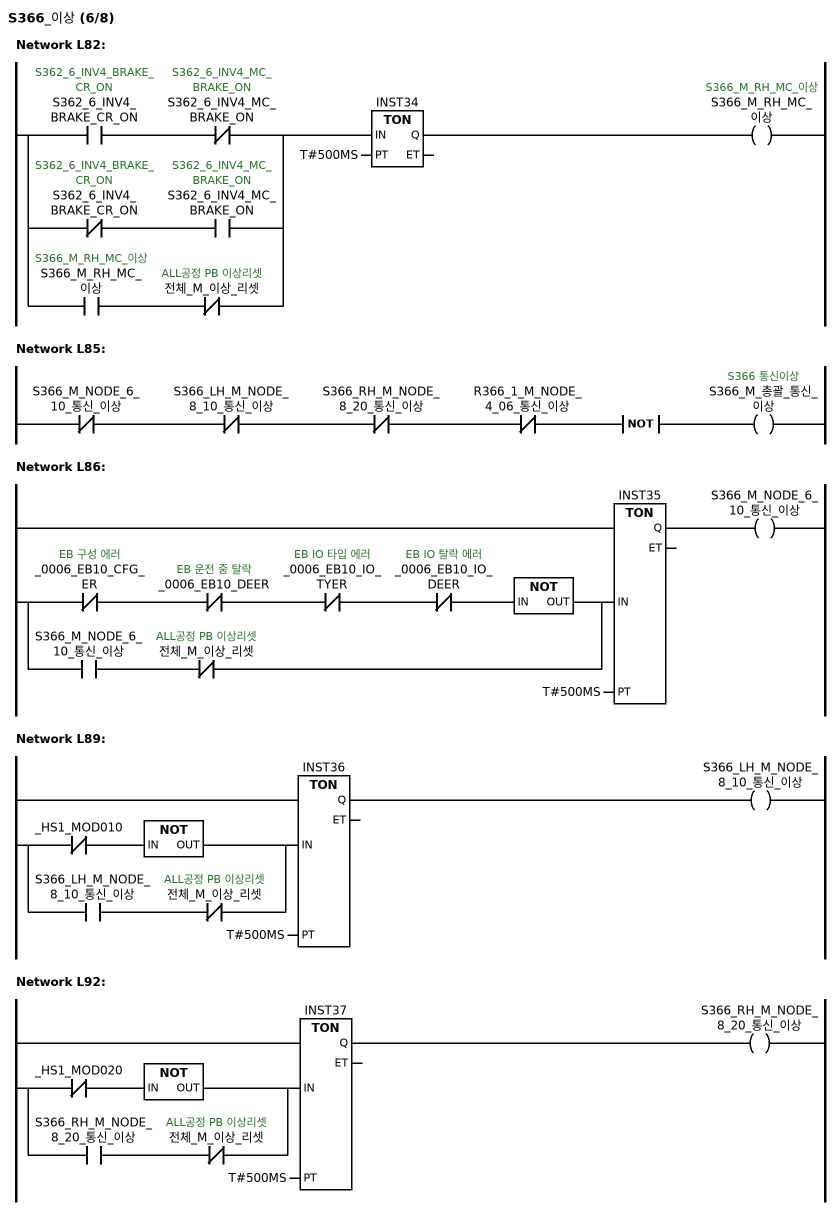
(* Rung L82 *)
INST34(IN := (S362_6_INV4_BRAKE_CR_ON AND NOT S362_6_INV4_MC_BRAKE_ON) OR (NOT S362_6_INV4_BRAKE_CR_ON AND S362_6_INV4_MC_BRAKE_ON) OR (S366_M_RH_MC_이상 AND NOT 전체_M_이상_리셋), PT := T#500MS);
S366_M_RH_MC_이상 := INST34.Q;
(* Rung L85 *)
S366_M_총괄_통신_이상 := NOT (NOT S366_M_NODE_6_10_통신_이상 AND NOT S366_LH_M_NODE_8_10_통신_이상 AND NOT S366_RH_M_NODE_8_20_통신_이상 AND NOT R366_1_M_NODE_4_06_통신_이상);
(* Rung L86 *)
INST35(IN := (NOT (NOT _0006_EB10_CFG_ER AND NOT _0006_EB10_DEER AND NOT _0006_EB10_IO_TYER AND NOT _0006_EB10_IO_DEER)) OR (S366_M_NODE_6_10_통신_이상 AND NOT 전체_M_이상_리셋), PT := T#500MS);
S366_M_NODE_6_10_통신_이상 := INST35.Q;
(* Rung L89 *)
INST36(IN := (NOT (NOT _HS1_MOD010)) OR (S366_LH_M_NODE_8_10_통신_이상 AND NOT 전체_M_이상_리셋), PT := T#500MS);
S366_LH_M_NODE_8_10_통신_이상 := INST36.Q;
(* Rung L92 *)
INST37(IN := (NOT (NOT _HS1_MOD020)) OR (S366_RH_M_NODE_8_20_통신_이상 AND NOT 전체_M_이상_리셋), PT := T#500MS);
S366_RH_M_NODE_8_20_통신_이상 := INST37.Q;

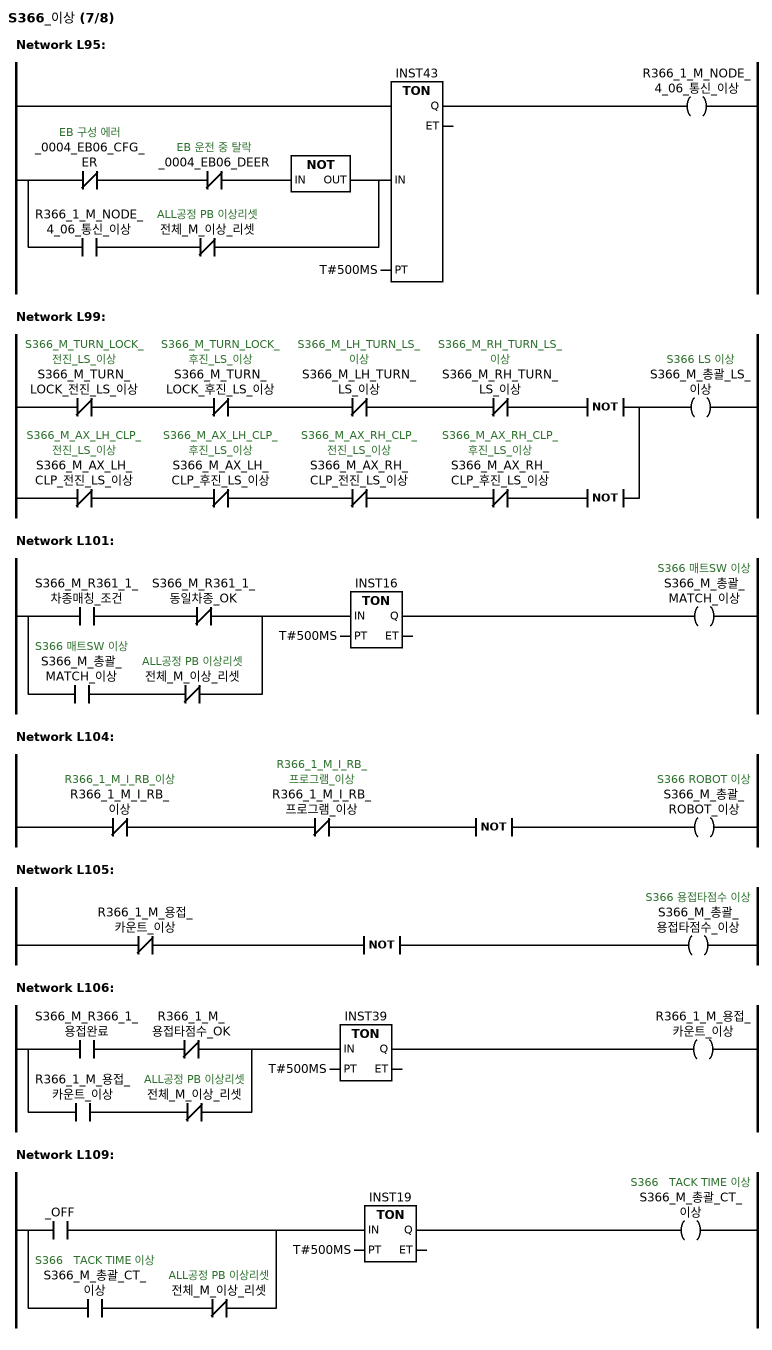
(* Rung L95 *)
INST43(IN := (NOT (NOT _0004_EB06_CFG_ER AND NOT _0004_EB06_DEER)) OR (R366_1_M_NODE_4_06_통신_이상 AND NOT 전체_M_이상_리셋), PT := T#500MS);
R366_1_M_NODE_4_06_통신_이상 := INST43.Q;
(* Rung L99 *)
S366_M_총괄_LS_이상 := NOT (NOT S366_M_TURN_LOCK_전진_LS_이상 AND NOT S366_M_TURN_LOCK_후진_LS_이상 AND NOT S366_M_LH_TURN_LS_이상 AND NOT S366_M_RH_TURN_LS_이상) OR NOT (NOT S366_M_AX_LH_CLP_전진_LS_이상 AND NOT S366_M_AX_LH_CLP_후진_LS_이상 AND NOT S366_M_AX_RH_CLP_전진_LS_이상 AND NOT S366_M_AX_RH_CLP_후진_LS_이상);
(* Rung L101 *)
INST16(IN := (S366_M_R361_1_차종매칭_조건 AND NOT S366_M_R361_1_동일차종_OK) OR (S366_M_총괄_MATCH_이상 AND NOT 전체_M_이상_리셋), PT := T#500MS);
S366_M_총괄_MATCH_이상 := INST16.Q;
(* Rung L104 *)
S366_M_총괄_ROBOT_이상 := NOT (NOT R366_1_M_I_RB_이상 AND NOT R366_1_M_I_RB_프로그램_이상);
(* Rung L105 *)
S366_M_총괄_용접타점수_이상 := R366_1_M_용접_카운트_이상;
(* Rung L106 *)
INST39(IN := (S366_M_R366_1_용접완료 AND NOT R366_1_M_용접타점수_OK) OR (R366_1_M_용접_카운트_이상 AND NOT 전체_M_이상_리셋), PT := T#500MS);
R366_1_M_용접_카운트_이상 := INST39.Q;
(* Rung L109 *)
INST19(IN := _OFF OR (S366_M_총괄_CT_이상 AND NOT 전체_M_이상_리셋), PT := T#500MS);
S366_M_총괄_CT_이상 := INST19.Q;

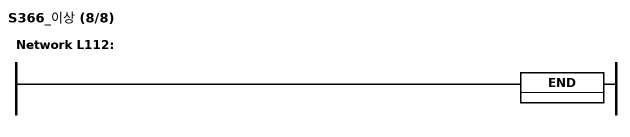
(* Rung L112 *)
END();
END_PROGRAM

PROGRAM S367_유틸리티 (* task: 스캔 프로그램 *)
VAR_EXTERNAL
    EGIS_CWS : BOOL;
    HOP_PBL_365_8_자동_운전 : BOOL; (* AT %MW87500.7 *) (* HOP_PBL_365_8_자동_운전 *)
    HOP_PBL_운전준비_ON : BOOL; (* AT %MW87500.0 *) (* HOP_PBL_운전준비_ON *)
    HOP_SSP_365_8_수동_선택 : BOOL; (* AT %MW87500.6 *) (* HOP_SSP_365_8_수동_선택 *)
    HOP_SSP_365_8_자동_선택 : BOOL; (* AT %MW87500.5 *) (* HOP_SSP_365_8_자동_선택 *)
    MCP_PBL_365_8_자동_운전 : BOOL; (* AT %MW87630.7 *) (* MCP PBL 365~8 자동기동 *)
    MCP_PBL_운전준비_ON : BOOL; (* AT %MW87630.0 *) (* MCP_PBL_운전준비_ON *)
    MCP_SPB_작업완료_RESET : BOOL; (* AT %MW87631.6 *) (* MCP_SPB_작업완료_RESET *)
    MCP_SPB_작업완료_SET : BOOL; (* AT %MW87631.7 *) (* MCP_SPB_작업완료_SET *)
    MCP_SSP_365_8_수동_선택 : BOOL; (* AT %MW87630.5 *) (* MCP_SSP_365_8_수동_선택 *)
    MCP_SSP_365_8_자동_선택 : BOOL; (* AT %MW87630.6 *) (* MCP_SSP_365_8_자동_선택 *)
    R361_1_M_I_RB_3차_작업완료 : BOOL; (* AT %MW20011.4 *) (* R361_1_M_I_RB_3차_작업완료 *)
    R361_1_M_I_RB_5차_작업완료 : BOOL; (* AT %MW20011.6 *) (* R361_1_M_I_RB_5차_작업완료 *)
    R361_1_M_I_RB_6차_작업완료 : BOOL; (* AT %MW20011.7 *) (* R361_1_M_I_RB_6차_작업완료 *)
    R361_1_M_I_RB_간섭무_1 : BOOL; (* AT %MW20012.0 *) (* R361_1_M_I_RB_간섭무_1 *)
    R361_1_M_I_RB_원위치 : BOOL; (* AT %MW20010.3 *) (* R361_1_M_I_RB_원위치 *)
    R366_1_M_I_RB_1차_작업완료 : BOOL; (* AT %MW20061.2 *) (* R366_1_M_I_RB_1차_작업완료 *)
    R366_1_M_I_RB_2차_작업완료 : BOOL; (* AT %MW20061.3 *) (* R366_1_M_I_RB_2차_작업완료 *)
    R366_1_M_I_RB_간섭무_1 : BOOL; (* AT %MW20062.0 *) (* R366_1_M_I_RB_간섭무_1 *)
    R366_1_M_I_RB_원위치 : BOOL; (* AT %MW20060.3 *) (* R366_1_M_I_RB_원위치 *)
    R369_1_M_I_RB_1차_작업완료 : BOOL; (* AT %MW20081.2 *) (* R369_1_M_I_RB_1차_작업완료 *)
    R369_1_M_I_RB_간섭무_1 : BOOL; (* AT %MW20082.0 *) (* R369_1_M_I_RB_간섭무_1 *)
    R369_1_M_I_RB_원위치 : BOOL; (* AT %MW20080.3 *) (* R369_1_M_I_RB_원위치 *)
    S367_PRS_AX_LH_ROOF_FRT_CHK : BOOL; (* AT %MW86212.0 *) (* S367_PRS_AX_LH_ROOF_FRT_CHK *)
    S367_PRS_AX_LH_ROOF_RR_CHK : BOOL; (* AT %MW86212.1 *) (* S367_PRS_AX_LH_ROOF_RR_CHK *)
    S367_PRS_AX_RH_ROOF_FRT_CHK : BOOL; (* AT %MW86202.0 *) (* S367_PRS_AX_RH_ROOF_FRT_CHK *)
    S367_PRS_AX_RH_ROOF_RR_CHK : BOOL; (* AT %MW86202.1 *) (* S367_PRS_AX_RH_ROOF_RR_CHK *)
END_VAR
VAR_EXTERNAL RETAIN
    HMI_M_선택_MOD_S367 : BOOL; (* AT %MW6.5 *) (* HMI M 선택 MOD S367 *)
    R361_1_M_차종6_썬루프 : BOOL; (* AT %MW10003.4 *) (* R361 1 M 차종6 썬루프 *)
    R361_1_M_차종6_일반루프 : BOOL; (* AT %MW10003.3 *) (* R361 1 M 차종6 일반루프 *)
    S362_M_총괄_이상 : BOOL; (* AT %MW1009.0 *) (* S362_M_총괄_이상 *)
    S366_M_공정_차종_무 : BOOL; (* AT %MW3002.1 *) (* S366_M_공정_차종_무 *)
    S366_M_공정_차종_유 : BOOL; (* AT %MW3002.0 *) (* S366_M_공정_차종_유 *)
    S366_M_작업완료_SET_PLS : BOOL; (* AT %MW3000.8 *) (* S366 M 작업완료 SET PLS *)
    S366_M_작업완료_리셋_PLS : BOOL; (* AT %MW3000.9 *) (* S366 M 작업완료 리셋 PLS *)
    S366_M_차종1_AX : BOOL; (* AT %MW10161.0 *) (* S366 M 차종1 AX *)
    S366_M_차종1_B : BOOL; (* AT %MW10161.1 *) (* S366 M 차종1 B *)
    S366_M_차종1_C : BOOL; (* AT %MW10161.2 *) (* S366 M 차종1 C *)
    S366_M_차종1_D : BOOL; (* AT %MW10161.3 *) (* S366 M 차종1 D *)
    S367_M_369_1_언로딩가능 : BOOL; (* AT %MW3504.10 *)
    S367_M_BYPASS_보조 : BOOL; (* AT %MW3503.15 *) (* S367 M BYPASS 보조 *)
    S367_M_LH_AX_CLAMP_전진단 : BOOL; (* AT %MW3602.3 *) (* S367_M_LH_AX_CLAMP_전진단 *)
    S367_M_LH_AX_CLAMP_후진단 : BOOL; (* AT %MW3602.4 *) (* S367_M_LH_AX_CLAMP_후진단 *)
    S367_M_LH_AX_LATCH_전진단 : BOOL; (* AT %MW3600.3 *) (* S367_M_LH_AX_LATCH_전진단 *)
    S367_M_LH_AX_LATCH_후진단 : BOOL; (* AT %MW3600.4 *) (* S367_M_LH_AX_LATCH_후진단 *)
    S367_M_LH_AX_SR_LAT_전진단 : BOOL; (* AT %MW3601.3 *) (* S367_M_LH_AX_SR_LAT_전진단 *)
    S367_M_LH_AX_SR_LAT_후진단 : BOOL; (* AT %MW3601.4 *) (* S367_M_LH_AX_SR_LAT_후진단 *)
    S367_M_R361_1_로딩가능 : BOOL; (* AT %MW3504.8 *)
    S367_M_R361_1_로딩완료 : BOOL; (* AT %MW3501.1 *)
    S367_M_R366_1_용접가능 : BOOL; (* AT %MW3504.9 *)
    S367_M_R366_1_용접완료 : BOOL; (* AT %MW3501.2 *)
    S367_M_R369_1_언로딩완료 : BOOL; (* AT %MW3501.3 *)
    S367_M_RH_AX_CLAMP_전진단 : BOOL; (* AT %MW3610.3 *) (* S367_M_RH_AX_CLAMP_전진단 *)
    S367_M_RH_AX_CLAMP_후진단 : BOOL; (* AT %MW3610.4 *) (* S367_M_RH_AX_CLAMP_후진단 *)
    S367_M_RH_AX_LATCH_전진단 : BOOL; (* AT %MW3608.3 *) (* S367_M_RH_AX_LATCH_전진단 *)
    S367_M_RH_AX_LATCH_후진단 : BOOL; (* AT %MW3608.4 *) (* S367_M_RH_AX_LATCH_후진단 *)
    S367_M_RH_AX_SR_LAT_전진단 : BOOL; (* AT %MW3609.3 *) (* S367_M_RH_AX_SR_LAT_전진단 *)
    S367_M_RH_AX_SR_LAT_후진단 : BOOL; (* AT %MW3609.4 *) (* S367_M_RH_AX_SR_LAT_후진단 *)
    S367_M_SEQ : WORD; (* AT %MW10180 *) (* S367 M SEQ *)
    S367_M_공정_FRT_제품감지_무 : BOOL; (* AT %MW3501.8 *)
    S367_M_공정_FRT_제품감지_유 : BOOL; (* AT %MW3501.7 *)
    S367_M_공정_RR_제품감지_무 : BOOL; (* AT %MW3501.10 *)
    S367_M_공정_RR_제품감지_유 : BOOL; (* AT %MW3501.9 *)
    S367_M_공정_불간섭 : BOOL; (* AT %MW3504.1 *) (* S367_M_공정_불간섭 *)
    S367_M_공정_원위치 : BOOL; (* AT %MW3504.0 *) (* S367_M_공정_원위치 *)
    S367_M_공정_제품감지_무 : BOOL; (* AT %MW3501.6 *) (* S367_M_공정_제품감지_무 *)
    S367_M_공정_제품감지_유 : BOOL; (* AT %MW3501.5 *) (* S367_M_공정_제품감지_유 *)
    S367_M_공정_차종_무 : BOOL; (* AT %MW3502.1 *) (* S367_M_공정_차종_무 *)
    S367_M_공정_차종_유 : BOOL; (* AT %MW3502.0 *) (* S367_M_공정_차종_유 *)
    S367_M_수동모드 : BOOL; (* AT %MW3500.3 *) (* S367 선택 수동모드 *)
    S367_M_운전준비_ON : BOOL; (* AT %MW3500.0 *) (* S367 운전준비 ON *)
    S367_M_자동_START : BOOL; (* AT %MW3500.5 *) (* S367 자동운전중 *)
    S367_M_자동_운전중 : BOOL; (* AT %MW3500.4 *) (* S367 자동운전중 *)
    S367_M_자동모드 : BOOL; (* AT %MW3500.1 *) (* S367 선택 자동모드 *)
    S367_M_작업_완료 : BOOL; (* AT %MW3501.0 *) (* S367_M_작업_완료 *)
    S367_M_작업완료_SET_PLS : BOOL; (* AT %MW3500.8 *) (* S367 M 작업완료 SET PLS *)
    S367_M_작업완료_리셋_PLS : BOOL; (* AT %MW3500.9 *) (* S367 M 작업완료 리셋 PLS *)
    S367_M_차종1_AX : BOOL; (* AT %MW10181.0 *) (* S367 M 차종1 AX *)
    S367_M_차종1_B : BOOL; (* AT %MW10181.1 *) (* S367 M 차종1 B *)
    S367_M_차종1_C : BOOL; (* AT %MW10181.2 *) (* S367 M 차종1 C *)
    S367_M_차종1_D : BOOL; (* AT %MW10181.3 *) (* S367 M 차종1 D *)
    S367_M_차종1_E : BOOL; (* AT %MW10181.4 *) (* S367 M 차종1 E *)
    S367_M_차종1_F : BOOL; (* AT %MW10181.5 *) (* S367 M 차종1 F *)
    S367_M_차종1_G : BOOL; (* AT %MW10181.6 *) (* S367 M 차종1 G *)
    S367_M_차종1_H : BOOL; (* AT %MW10181.7 *) (* S367 M 차종1 H *)
    S367_M_차종2_3DR : BOOL; (* AT %MW10181.8 *) (* S367 M 차종2 3DR *)
    S367_M_차종2_4DR : BOOL; (* AT %MW10181.9 *) (* S367 M 차종2 4DR *)
    S367_M_차종2_5DR : BOOL; (* AT %MW10181.10 *) (* S367 M 차종2 5DR *)
    S367_M_차종2_SP1 : BOOL; (* AT %MW10181.12 *) (* S367 M 차종2 SP1 *)
    S367_M_차종2_SP2 : BOOL; (* AT %MW10181.13 *) (* S367 M 차종2 SP2 *)
    S367_M_차종2_WGN : BOOL; (* AT %MW10181.11 *) (* S367 M 차종2 WGN *)
    S367_M_차종3_LHD : BOOL; (* AT %MW10181.14 *) (* S367 M 차종3 LHD *)
    S367_M_차종3_RHD : BOOL; (* AT %MW10181.15 *) (* S367 M 차종3 RHD *)
    S367_M_차종4_EEC : BOOL; (* AT %MW10182.3 *) (* S367 M 차종4 EEC *)
    S367_M_차종4_SP1 : BOOL; (* AT %MW10182.8 *) (* S367 M 차종4 SP1 *)
    S367_M_차종4_SP2 : BOOL; (* AT %MW10182.9 *) (* S367 M 차종4 SP2 *)
    S367_M_차종4_SP3 : BOOL; (* AT %MW10182.11 *) (* S367 M 차종4 SP3 *)
    S367_M_차종4_SP4 : BOOL; (* AT %MW10182.12 *) (* S367 M 차종4 SP4 *)
    S367_M_차종4_SP5 : BOOL; (* AT %MW10182.13 *) (* S367 M 차종4 SP5 *)
    S367_M_차종4_SP6 : BOOL; (* AT %MW10182.14 *) (* S367 M 차종4 SP6 *)
    S367_M_차종4_SP7 : BOOL; (* AT %MW10182.15 *) (* S367 M 차종4 SP7 *)
    S367_M_차종4_내수 : BOOL; (* AT %MW10182.0 *) (* S367 M 차종4 내수 *)
    S367_M_차종4_러시아 : BOOL; (* AT %MW10182.10 *) (* S367 M 차종4 러시아 *)
    S367_M_차종4_북미 : BOOL; (* AT %MW10182.2 *) (* S367 M 차종4 북미 *)
    S367_M_차종4_브라질 : BOOL; (* AT %MW10182.7 *) (* S367 M 차종4 브라질 *)
    S367_M_차종4_수출 : BOOL; (* AT %MW10182.1 *) (* S367 M 차종4 수출 *)
    S367_M_차종4_중국 : BOOL; (* AT %MW10182.6 *) (* S367 M 차종4 중국 *)
    S367_M_차종4_중동 : BOOL; (* AT %MW10182.5 *) (* S367 M 차종4 중동 *)
    S367_M_차종4_호주 : BOOL; (* AT %MW10182.4 *) (* S367 M 차종4 호주 *)
    S367_M_차종5_AT : BOOL; (* AT %MW10183.1 *) (* S367 M 차종5 AT *)
    S367_M_차종5_MT : BOOL; (* AT %MW10183.0 *) (* S367 M 차종5 MT *)
    S367_M_차종5_SP1 : BOOL; (* AT %MW10183.2 *) (* S367 M 차종5 SP1 *)
    S367_M_차종6_DSROOF : BOOL; (* AT %MW10183.6 *) (* S367 M 차종6 DSROOF *)
    S367_M_차종6_SP1 : BOOL; (* AT %MW10183.7 *) (* S367 M 차종6 SP1 *)
    S367_M_차종6_썬루프 : BOOL; (* AT %MW10183.4 *) (* S367 M 차종6 썬루프 *)
    S367_M_차종6_일반루프 : BOOL; (* AT %MW10183.3 *) (* S367 M 차종6 일반루프 *)
    S367_M_차종6_파노라마루프 : BOOL; (* AT %MW10183.5 *) (* S367 M 차종6 파노라마루프 *)
    S367_M_차종7_DSL : BOOL; (* AT %MW10183.9 *) (* S367 M 차종7 DSL *)
    S367_M_차종7_GSL : BOOL; (* AT %MW10183.8 *) (* S367 M 차종7 GSL *)
    S367_M_차종7_SP1 : BOOL; (* AT %MW10183.10 *) (* S367 M 차종7 SP1 *)
    S367_M_차종7_SP2 : BOOL; (* AT %MW10183.11 *) (* S367 M 차종7 SP2 *)
    S367_M_차종7_SP3 : BOOL; (* AT %MW10183.12 *) (* S367 M 차종7 SP3 *)
    S367_M_차종7_SP4 : BOOL; (* AT %MW10183.13 *) (* S367 M 차종7 SP4 *)
    S367_M_차종7_SP5 : BOOL; (* AT %MW10183.14 *) (* S367 M 차종7 SP5 *)
    S367_M_차종7_SP6 : BOOL; (* AT %MW10183.15 *) (* S367 M 차종7 SP6 *)
    S367_M_차종8_2WD : BOOL; (* AT %MW10184.0 *) (* S367 M 차종8 2WD *)
    S367_M_차종8_4WD : BOOL; (* AT %MW10184.1 *) (* S367 M 차종8 4WD *)
    S367_M_차종8_SP1 : BOOL; (* AT %MW10184.2 *) (* S367 M 차종8 SP1 *)
    S367_M_차종9_MPI : BOOL; (* AT %MW10184.3 *) (* S367 M 차종9 MPI *)
    S367_M_차종9_SP1 : BOOL; (* AT %MW10184.5 *) (* S367 M 차종9 SP1 *)
    S367_M_차종9_SP10 : BOOL; (* AT %MW10184.14 *) (* S367 M 차종9 SP10 *)
    S367_M_차종9_SP11 : BOOL; (* AT %MW10184.15 *) (* S367 M 차종9 SP11 *)
    S367_M_차종9_SP2 : BOOL; (* AT %MW10184.6 *) (* S367 M 차종9 SP2 *)
    S367_M_차종9_SP3 : BOOL; (* AT %MW10184.7 *) (* S367 M 차종9 SP3 *)
    S367_M_차종9_SP4 : BOOL; (* AT %MW10184.8 *) (* S367 M 차종9 SP4 *)
    S367_M_차종9_SP5 : BOOL; (* AT %MW10184.9 *) (* S367 M 차종9 SP5 *)
    S367_M_차종9_SP6 : BOOL; (* AT %MW10184.10 *) (* S367 M 차종9 SP6 *)
    S367_M_차종9_SP7 : BOOL; (* AT %MW10184.11 *) (* S367 M 차종9 SP7 *)
    S367_M_차종9_SP8 : BOOL; (* AT %MW10184.12 *) (* S367 M 차종9 SP8 *)
    S367_M_차종9_SP9 : BOOL; (* AT %MW10184.13 *) (* S367 M 차종9 SP9 *)
    S367_M_차종9_T_GDI : BOOL; (* AT %MW10184.4 *) (* S367 M 차종9 T GDI *)
    S367_M_차종_OPT1_R_RACK_무 : BOOL; (* AT %MW10185.3 *) (* S367 M 차종 OPT1 R RACK 무 *)
    S367_M_차종_OPT1_R_RACK_유 : BOOL; (* AT %MW10185.2 *) (* S367 M 차종 OPT1 R RACK 유 *)
    S367_M_차종_OPT1_S_REP_EATER_무 : BOOL; (* AT %MW10185.7 *) (* S367 M 차종 OPT1 S REP EATER 무 *)
    S367_M_차종_OPT1_S_REP_EATER_유 : BOOL; (* AT %MW10185.6 *) (* S367 M 차종 OPT1 S REP EATER 유 *)
    S367_M_차종_OPT1_VAN_무 : BOOL; (* AT %MW10185.9 *) (* S367 M 차종 OPT1 VAN 무 *)
    S367_M_차종_OPT1_VAN_유 : BOOL; (* AT %MW10185.8 *) (* S367 M 차종 OPT1 VAN 유 *)
    S367_M_차종_OPT1_슬라이딩_무 : BOOL; (* AT %MW10185.1 *) (* S367 M 차종 OPT1 슬라이딩 무 *)
    S367_M_차종_OPT1_슬라이딩_유 : BOOL; (* AT %MW10185.0 *) (* S367 M 차종 OPT1 슬라이딩 유 *)
    S367_M_차종_OPT1_폴딩_무 : BOOL; (* AT %MW10185.5 *) (* S367 M 차종 OPT1 폴딩 무 *)
    S367_M_차종_OPT1_폴딩_유 : BOOL; (* AT %MW10185.4 *) (* S367 M 차종 OPT1 폴딩 유 *)
    S367_M_차종_공대차 : BOOL; (* AT %MW10190.12 *) (* S367 M 차종 공대차 *)
    S367_M_차종_공차 : BOOL; (* AT %MW10190.10 *) (* S367 M 차종 공차 *)
    S367_M_차종_불량차 : BOOL; (* AT %MW10190.11 *) (* S367 M 차종 불량차 *)
    S367_M_총괄_이상 : BOOL; (* AT %MW3509.0 *) (* S367_M_총괄_이상 *)
    전체_M_GATE_자동기동 : BOOL; (* AT %MW308.1 *) (* 전체_M_자동_운전 *)
    전체_라인_M_총괄_SAFETY_이상 : BOOL; (* AT %MW300.2 *) (* ALL공정 SAFETY  이상총괄 *)
    전체_라인_M_총괄_공기압_이상 : BOOL; (* AT %MW300.3 *) (* ALL공정 공기압 이상총괄 *)
    전체_라인_M_총괄_비상정지_이상 : BOOL; (* AT %MW300.1 *) (* ALL공정 비상정지 이상총괄 *)
    전체_라인_M_총괄_이상 : BOOL; (* AT %MW300.0 *) (* ALL공정 총괄이상 *)
END_VAR
VAR
    S367_READY : TON;
    T367_AUTO : TON;
END_VAR
VAR
    _t1 : BOOL;
END_VAR

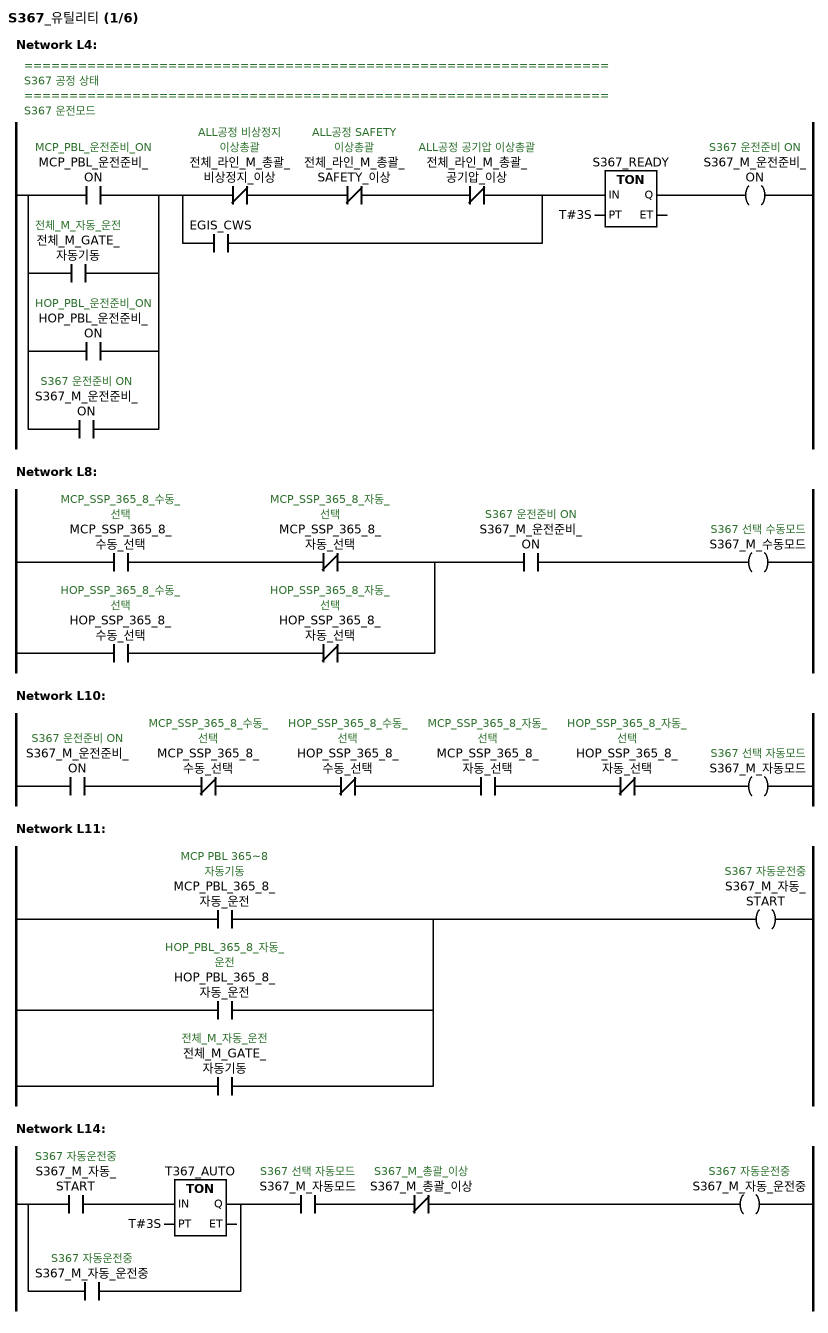
(* ================================================================= *)
(* S367 공정 상태 *)
(* ================================================================= *)
(* S367 운전모드 *)
(* Rung L4 *)
S367_READY(IN := (MCP_PBL_운전준비_ON OR 전체_M_GATE_자동기동 OR HOP_PBL_운전준비_ON OR S367_M_운전준비_ON) AND ((NOT 전체_라인_M_총괄_비상정지_이상 AND NOT 전체_라인_M_총괄_SAFETY_이상 AND NOT 전체_라인_M_총괄_공기압_이상) OR EGIS_CWS), PT := T#3S);
S367_M_운전준비_ON := S367_READY.Q;
(* Rung L8 *)
S367_M_수동모드 := ((MCP_SSP_365_8_수동_선택 AND NOT MCP_SSP_365_8_자동_선택) OR (HOP_SSP_365_8_수동_선택 AND NOT HOP_SSP_365_8_자동_선택)) AND S367_M_운전준비_ON;
(* Rung L10 *)
S367_M_자동모드 := S367_M_운전준비_ON AND NOT MCP_SSP_365_8_수동_선택 AND NOT HOP_SSP_365_8_수동_선택 AND MCP_SSP_365_8_자동_선택 AND NOT HOP_SSP_365_8_자동_선택;
(* Rung L11 *)
S367_M_자동_START := MCP_PBL_365_8_자동_운전 OR HOP_PBL_365_8_자동_운전 OR 전체_M_GATE_자동기동;
(* Rung L14 *)
T367_AUTO(IN := S367_M_자동_START, PT := T#3S);
S367_M_자동_운전중 := (T367_AUTO.Q OR S367_M_자동_운전중) AND S367_M_자동모드 AND NOT S367_M_총괄_이상;

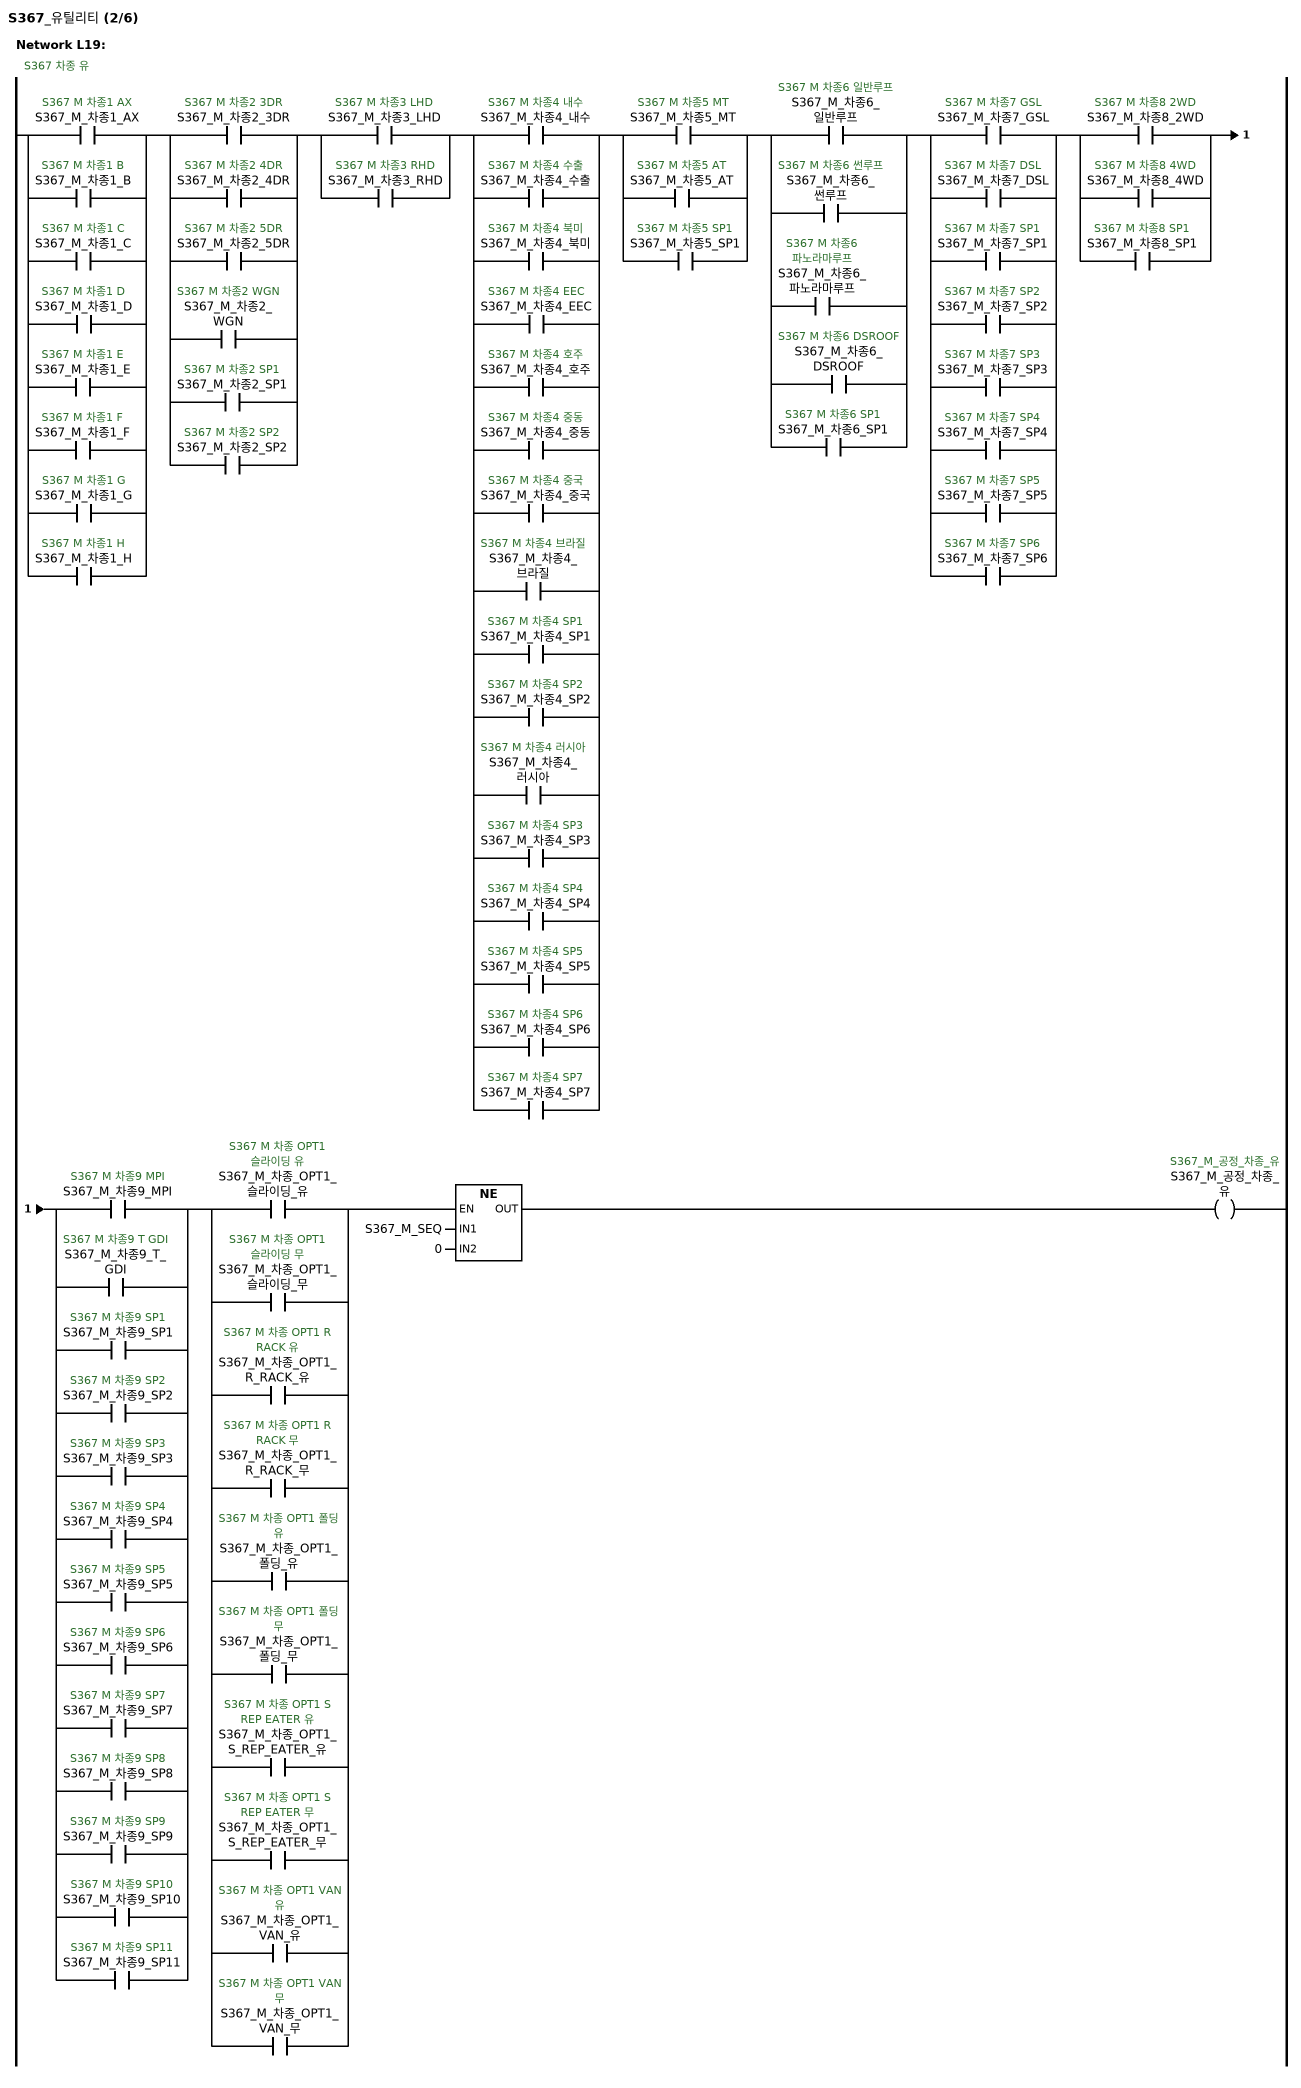
(* S367 차종 유 *)
(* Rung L19 *)
IF (S367_M_차종1_AX OR S367_M_차종1_B OR S367_M_차종1_C OR S367_M_차종1_D OR S367_M_차종1_E OR S367_M_차종1_F OR S367_M_차종1_G OR S367_M_차종1_H) AND (S367_M_차종2_3DR OR S367_M_차종2_4DR OR S367_M_차종2_5DR OR S367_M_차종2_WGN OR S367_M_차종2_SP1 OR S367_M_차종2_SP2) AND (S367_M_차종3_LHD OR S367_M_차종3_RHD) AND (S367_M_차종4_내수 OR S367_M_차종4_수출 OR S367_M_차종4_북미 OR S367_M_차종4_EEC OR S367_M_차종4_호주 OR S367_M_차종4_중동 OR S367_M_차종4_중국 OR S367_M_차종4_브라질 OR S367_M_차종4_SP1 OR S367_M_차종4_SP2 OR S367_M_차종4_러시아 OR S367_M_차종4_SP3 OR S367_M_차종4_SP4 OR S367_M_차종4_SP5 OR S367_M_차종4_SP6 OR S367_M_차종4_SP7) AND (S367_M_차종5_MT OR S367_M_차종5_AT OR S367_M_차종5_SP1) AND (S367_M_차종6_일반루프 OR S367_M_차종6_썬루프 OR S367_M_차종6_파노라마루프 OR S367_M_차종6_DSROOF OR S367_M_차종6_SP1) AND (S367_M_차종7_GSL OR S367_M_차종7_DSL OR S367_M_차종7_SP1 OR S367_M_차종7_SP2 OR S367_M_차종7_SP3 OR S367_M_차종7_SP4 OR S367_M_차종7_SP5 OR S367_M_차종7_SP6) AND (S367_M_차종8_2WD OR S367_M_차종8_4WD OR S367_M_차종8_SP1) AND (S367_M_차종9_MPI OR S367_M_차종9_T_GDI OR S367_M_차종9_SP1 OR S367_M_차종9_SP2 OR S367_M_차종9_SP3 OR S367_M_차종9_SP4 OR S367_M_차종9_SP5 OR S367_M_차종9_SP6 OR S367_M_차종9_SP7 OR S367_M_차종9_SP8 OR S367_M_차종9_SP9 OR S367_M_차종9_SP10 OR S367_M_차종9_SP11) AND (S367_M_차종_OPT1_슬라이딩_유 OR S367_M_차종_OPT1_슬라이딩_무 OR S367_M_차종_OPT1_R_RACK_유 OR S367_M_차종_OPT1_R_RACK_무 OR S367_M_차종_OPT1_폴딩_유 OR S367_M_차종_OPT1_폴딩_무 OR S367_M_차종_OPT1_S_REP_EATER_유 OR S367_M_차종_OPT1_S_REP_EATER_무 OR S367_M_차종_OPT1_VAN_유 OR S367_M_차종_OPT1_VAN_무) THEN
    _t1 := S367_M_SEQ <> 0;
END_IF;
S367_M_공정_차종_유 := _t1;

